//	Safety.GetDiagnostics(AddError:= AddError, a_ActiveEvents := a_ActiveEvents, w_index := w_errorindex);
//	Main_Fast.PowerMonitor.GetDiagnostics(AddError:= AddError, a_ActiveEvents := a_ActiveEvents, w_index := w_errorindex);
//	Main_Fast.InternalPowerSupply.GetDiagnostics(AddError:= AddError, a_ActiveEvents := a_ActiveEvents, w_index := w_errorindex);
//	Main_Fast.NeutralTransformer.GetDiagnostics(AddError:= AddError, a_ActiveEvents := a_ActiveEvents, w_index := w_errorindex);
//	Main_Fast.PowerStack.GetDiagnostics(AddError := AddError, a_ActiveEvents := a_ActiveEvents, w_index := w_errorindex);
//Main_Fast.Protectionsystems.GetDiagnostics(AddError := AddError, a_ActiveEvents := a_ActiveEvents, w_index := w_errorindex);
END_IF

//If larger than 0, error is existing
b_errorActive := GVL.b_NormalShutdownActive OR GVL.b_QuickshutdownActive OR GVL.b_EmergencyShutdownActive;

METHOD PUBLIC LimitTrigger
VAR_INPUT
	r_HighLimit				: REAL := 0;
	r_HighWarning			: REAL := 0;
	b_HighEnable			: BOOL := FALSE;
	r_LowLimit				: REAL := 0;
	r_LowWarning			: REAL := 0;
	b_LowEnable				: BOOL := FALSE;
	r_Hysteresis			: REAL := 0;
END_VAR

VAR_IN_OUT
	r_In					: REAL;
END_VAR

VAR_OUTPUT
	b_Warning				: BOOL;
	b_Fault					: BOOL;
END_VAR
IF b_HighEnable THEN
	IF r_IN >= r_HighLimit THEN
		b_Fault := TRUE;
	ELSIF r_IN < (r_HighLimit - r_Hysteresis) THEN
		b_fault := FALSE;
	END_IF
	IF r_IN >= r_HighWarning THEN
		b_warning := TRUE;
	ELSIF r_IN < (r_HighWarning - r_Hysteresis) THEN
		b_warning := FALSE;
	END_IF

END_IF

IF b_LowEnable THEN
	IF r_IN <= r_LowLimit THEN
		b_fault := TRUE;
	ELSIF r_IN > (r_LowLimit + r_Hysteresis) THEN
		b_fault := FALSE;
	END_IF
	IF r_IN <= r_LowWarning THEN
		b_warning := TRUE;
	ELSIF r_IN > (r_LowWarning + r_Hysteresis) THEN
		b_warning:= FALSE;
	END_IF
END_IF
END_METHOD

END_PROGRAM

// ---- POUs/ErrorHandling/FB_AddErrorST.TcPOU
FUNCTION_BLOCK FB_AddErrorST
VAR_INPUT
	in_b_ErrorTrig				: BOOL;
	in_t_TriggerTime			: TIME := T#0S;
	in_b_AutoClear				: BOOL := FALSE;
	in_e_ErrAckAccess			: eErrAckAccess := eErrAckAccess.VDL; //default full access required
	w_ID						: WORD;
	s_message					: STRING;
	e_sev						: eSeverity;
END_VAR
VAR_IN_OUT
	out_st_Error 				: ST_ErrorStruct;
END_VAR

VAR_OUTPUT
	b_out						: BOOL;
END_VAR

VAR
	sr_ErrorActive				: SR;
	bIsInitialized 				: BOOL := FALSE;	
	ton_FaultTriggerTime		: TON;
	rTRIG_Fault					: R_TRIG;
	fTRIG_Fault					: F_TRIG;
	rTRIG_Clear					: R_TRIG;
	
	
	i_Counter				: INT; 
END_VAR

IF NOT bIsInitialized THEN
    // The code that you want to be executed at the first cycle
		out_st_Error.s_ID		:= TO_STRING(w_ID);	
		out_st_Error.s_Message	:= TO_STRING(s_Message);
		out_st_Error.s_Severity	:= TO_STRING(e_Sev);
END_IF

ton_FaultTriggerTime(IN:= in_b_ErrorTrig, PT:= in_t_TriggerTime);
sr_ErrorActive(SET1:= ton_FaultTriggerTime.Q, Q1=>out_st_error.b_ErrorActive);
b_out := sr_ErrorActive.Q1;

sr_ErrorActive.RESET := SEL( errorhandling.e_access>=in_e_ErrAckAccess,0,Errorhandling.b_ResetError);

CASE e_sev OF
		eSeverity.Warning 			: GVL.b_WarningActive := b_out;
		eSeverity.Normalshutdown 	: GVL.b_NormalshutdownActive := b_out;
		eSeverity.Quickshutdown 	: GVL.b_QuickShutdownActive := b_out;
		eSeverity.EmergencyShutdown	: GVL.b_EmergencyShutdownActive := b_out;
END_CASE


//CLEARING EVENTS
rTRIG_Fault(CLK:= b_out);
fTRIG_Fault(CLK:= b_out);
rTRIG_Clear(CLK:= ErrorHandling.b_ClearEvents OR SEL(in_b_autoClear,FALSE, errorhandling.ton_AutoResetClear.Q) );

IF rTRIG_Clear.Q AND NOT b_out THEN
	out_st_Error.s_DateError 	:= '';
	out_st_Error.s_TimeError 	:= '';
	out_st_Error.s_TimeCleared	:= '';
END_IF

IF rTRIG_Fault.Q THEN
	out_st_Error.s_DateError := GVL.s_SystemDate;
	out_st_Error.s_TimeError := GVL.s_SystemTime;
	out_st_Error.s_TimeCleared	:= '';
	
ELSIF fTrig_Fault.Q THEN
	out_st_Error.s_TimeCleared	:= GVL.s_SystemTime;
END_IF

bIsInitialized := TRUE;

END_FUNCTION_BLOCK

// ---- POUs/FunctionBlocks/fbDwordToReal.TcPOU
FUNCTION_BLOCK fbDwordToReal
VAR_INPUT
	in_B0					: BYTE ;
	in_B1					: BYTE ;
	in_B2					: BYTE ;
	in_B3					: BYTE ;
	in_r_Res				: REAL ;
	in_i_Offset				: INT ;
END_VAR
VAR_OUTPUT
	out_r_Value				: REAL ;
END_VAR
VAR
	di_AddedValue			: DINT;
	r_Signed				: REAL;
	r_ResolutionResolved	: REAL;
END_VAR

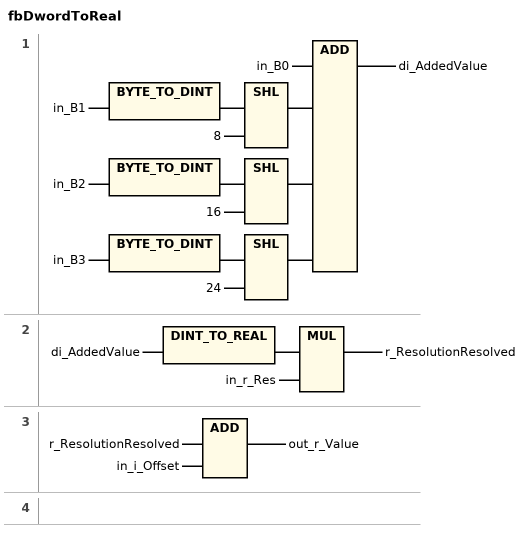
// NETWORK 1
di_AddedValue := in_B0 + SHL(BYTE_TO_DINT(in_B1), 8) + SHL(BYTE_TO_DINT(in_B2), 16) + SHL(BYTE_TO_DINT(in_B3), 24);

// NETWORK 2
r_ResolutionResolved := DINT_TO_REAL(di_AddedValue) * in_r_Res;

// NETWORK 3
out_r_Value := r_ResolutionResolved + in_i_Offset;

// NETWORK 4

END_FUNCTION_BLOCK

// ---- POUs/FunctionBlocks/fbRealToDWord.TcPOU
FUNCTION_BLOCK fbRealToDWord
VAR_INPUT
	in_r_Value				: REAL ;
	in_r_Res				: REAL ;
	in_i_Offset				: INT ;
END_VAR
VAR_OUTPUT
	out_B0					: BYTE ;
	out_B1					: BYTE ;
	out_B2					: BYTE ;
	out_B3					: BYTE ;
END_VAR
VAR
	dw_AddedValue			: DWORD;
	r_ResolutionResolved	: REAL;
	r_OffsetSolved			: REAL;
END_VAR

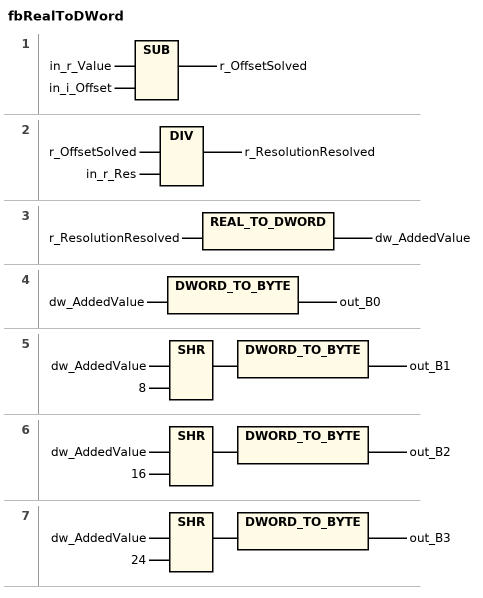
// NETWORK 1
r_OffsetSolved := in_r_Value - in_i_Offset;

// NETWORK 2
r_ResolutionResolved := r_OffsetSolved / in_r_Res;

// NETWORK 3
dw_AddedValue := REAL_TO_DWORD(r_ResolutionResolved);

// NETWORK 4
out_B0 := DWORD_TO_BYTE(dw_AddedValue);

// NETWORK 5
out_B1 := DWORD_TO_BYTE(SHR(dw_AddedValue, 8));

// NETWORK 6
out_B2 := DWORD_TO_BYTE(SHR(dw_AddedValue, 16));

// NETWORK 7
out_B3 := DWORD_TO_BYTE(SHR(dw_AddedValue, 24));

END_FUNCTION_BLOCK

// ---- POUs/FunctionBlocks/fbRealToWord.TcPOU
FUNCTION_BLOCK fbRealToWord
VAR_INPUT
	in_r_Value				: REAL ;
	in_r_Res				: REAL ;
	in_i_Offset				: INT ;
END_VAR
VAR_OUTPUT
	out_B0					: BYTE ;
	out_B1					: BYTE ;
END_VAR
VAR
	w_AddedValue			: WORD;
	r_ResolutionResolved	: REAL;
	r_OffsetSolved			: REAL;
END_VAR

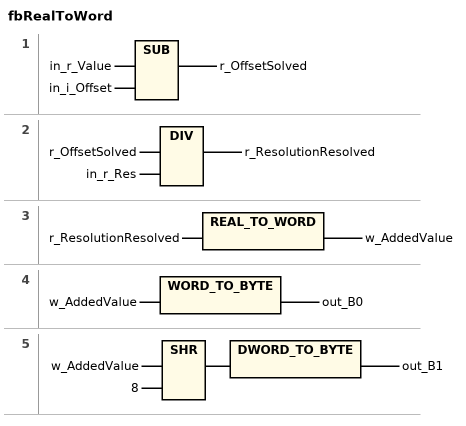
// NETWORK 1
r_OffsetSolved := in_r_Value - in_i_Offset;

// NETWORK 2
r_ResolutionResolved := r_OffsetSolved / in_r_Res;

// NETWORK 3
w_AddedValue := REAL_TO_WORD(r_ResolutionResolved);

// NETWORK 4
out_B0 := WORD_TO_BYTE(w_AddedValue);

// NETWORK 5
out_B1 := DWORD_TO_BYTE(SHR(w_AddedValue, 8));

END_FUNCTION_BLOCK

// ---- POUs/FunctionBlocks/fbWordToReal.TcPOU
FUNCTION_BLOCK fbWordToReal
VAR_INPUT
	in_B0					: BYTE ;
	in_B1					: BYTE ;
	in_r_Res				: REAL ;
	in_i_Offset				: INT ;
END_VAR
VAR_OUTPUT
	out_r_Value				: REAL ;
END_VAR
VAR
	dw_AddedValue			: DWORD;
	r_ResolutionResolved	: REAL;
END_VAR

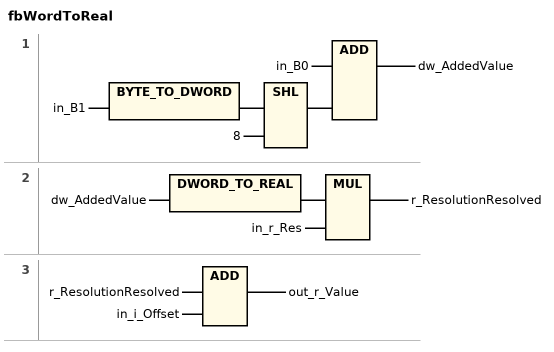
// NETWORK 1
dw_AddedValue := in_B0 + SHL(BYTE_TO_DWORD(in_B1), 8);

// NETWORK 2
r_ResolutionResolved := DWORD_TO_REAL(dw_AddedValue) * in_r_Res;

// NETWORK 3
out_r_Value := r_ResolutionResolved + in_i_Offset;

END_FUNCTION_BLOCK

// ---- POUs/MonitoringControl/FB_ControlManager.TcPOU
FUNCTION_BLOCK FB_ControlManager

VAR_OUTPUT PERSISTENT
	Hardsettings_persistent					: ST_HardSettings; 
	Softsettings_persistent					: ST_Softsettings;
END_VAR

VAR_OUTPUT
	control									: ST_ControlVars;
	Operation								: ST_OperationVars;
END_VAR

VAR
	IoT							: FB_ControlSource_IoT;	
	PNController				: FB_PNController;
	{ attribute 'TcHmiSymbol.Show' }
	b_SettingsChanged			: BOOL;				
END_VAR

VAR_IN_OUT CONSTANT
	{ attribute 'TcHmiSymbol.Hide' }
	monitor						: ST_SystemControl_FromSystem;
END_VAR

//instantiate fbs 
hmi(monitor:=monitor, PLCsettingsHard:= Hardsettings_persistent, PLCsettingsSoft :=SoftSettings_persistent);
PNController(monitor := monitor);
Iot(monitor:=monitor);

ControlSourceSelector();



//refresh HMI data --> future work make on change and asynchronous java in hmi

METHOD PROTECTED ControlSourceSelector

VAR_OUTPUT
	b_Busy					: BOOL;
	b_Error					: BOOL;
END_VAR

VAR
	
	softsettingsTemp				: ST_SoftSettings;
	controlTemp						: ST_ControlVars;
	
	rtrig_WritePersistent		: R_TRIG;
	fb_WritePersistentData		: WritePersistentData;
END_VAR
//Choosing the control source always requires the HMI
IF HMI.controlvars.control.b_ActivateSettings THEN
	Hardsettings_persistent.setup.e_ControlSource := HMI.Controlvars.hardSettings.setup.e_ControlSource;
END_IF


CASE Hardsettings_persistent.setup.e_ControlSource OF
	eControlSources.Local: // HMI
		softsettingsTemp 	:= HMI.controlvars.SoftSettings;
		Operation			:= HMI.controlvars.Operation;
	eControlSources.ExternalController: // HMI
		softsettingsTemp 	:= PnController.SoftSettings;
		Operation			:= PNController.Operation;	
		controlTemp			:= PNController.control;
	eControlSources.IoT:	//IOT
		softsettingsTemp 	:= IoT.SoftSettings; // Only local HMI can adjust recipe and thus persistent values.
		Operation			:= IoT.operation;
		controlTemp			:= IoT.control;
END_CASE

// WRITE PRIORITY DATA
control.b_start := HMI.controlvars.control.b_start OR controltemp.b_start;
control.b_Shutdown := HMI.controlvars.control.b_Shutdown OR controltemp.b_Shutdown;
control.b_ClearHistory := HMI.controlvars.control.b_ClearHistory OR controltemp.b_ClearHistory;
control.b_Reset := HMI.controlvars.control.b_Reset OR controltemp.b_Reset;
control.b_ActivateSettings := HMI.controlvars.control.b_ActivateSettings OR controltemp.b_ActivateSettings;
control.b_Reboot:= HMI.controlvars.control.b_Reboot OR controltemp.b_Reboot;
control.b_EMstop:= HMI.controlvars.control.b_EMstop OR controltemp.b_EMstop;
control.b_ResetVDL := HMI.controlvars.control.b_ResetVDL OR Iot.control.b_ResetVDL;


//WRITE PERSISTENT DATA
rtrig_WritePersistent(CLK:=HMI.controlvars.control.b_ActivateSettings);
IF rtrig_WritePersistent.Q THEN
	Hardsettings_persistent := HMI.controlvars.HardSettings;
	Softsettings_persistent	:= softsettingsTemp;
	fb_WritePersistentData(NETID := '', PORT:= 851, START:=TRUE, TMOUT := T#1S);
ELSE
	fb_WritePersistentData(START := FALSE);
END_IF

b_Busy := fb_WritePersistentData.BUSY;
b_Error := fb_WritePersistentData.ERR;
END_METHOD

END_FUNCTION_BLOCK

// ---- POUs/MonitoringControl/ProfinetController/FB_PNController.TcPOU
FUNCTION_BLOCK FB_PNController
VAR_OUTPUT
	{ attribute 'TcHmiSymbol.ShowRecursively' }
	control							: ST_ControlVars;	//1 module
	Operation						: ST_OperationVars;	//4 modules
	SoftSettings					: ST_SoftSettings;	//4 modules
	get								: ST_PNController_get;
END_VAR

VAR_IN_OUT CONSTANT
	{ attribute 'TcHmiSymbol.Hide' }
	monitor								: ST_SystemControl_FromSystem;
END_VAR

VAR
	CouplerState	AT %I*		:	WORD;	
	CouplerDiag		AT %I*		:	WORD;	

	GeneralInputs 	AT %I*		:	ST_PNInput_General;
	GeneralOutputs	AT %Q*		:	ST_PNOutput_General;
	
	BatteryInputs 	AT %I*		:	ST_PNInput_Battery;
	BatteryOutputs 	AT %Q*		:	ST_PNOutput_Battery;
	
	OutputFieldOutputs AT %Q*	:	ST_PNOutput_OutputField;
	
	InputFieldInputs	AT %I* 	:	ST_PNInput_InputField;
	InputFieldOutputs	AT %Q* 	:	ST_PNOutput_InputField;
	
	PowerStackInputs	AT %I* 	:	ST_PNInput_PowerStack;
	PowerStackOutputs	AT %Q* 	:	ST_PNOutput_PowerStack;	
	
	PeakShaveBoxInputs	AT %I* 	:	ST_PNInput_PeakShaveBox;
	PeakShaveBoxOutputs	AT %Q* 	:	ST_PNOutput_PeakShaveBox;
	
	ZPTOutputs			AT %Q* 	:	ST_PNOutput_ZPT;
	
END_VAR

VAR_INPUT
	b_enableControl	:	BOOL;
	b_enableMonitor	:	BOOL;
END_VAR


MapGeneralData	(Input := GeneralInputs, 		Output => Generaloutputs		);
MapBatteryData	(Input := BatteryInputs,		Output => BatteryOutputs		);
MapOutputField	(								Output => OutputFieldOutputs	);
MapInputField	(Input := InputFieldInputs, 	Output => InputFieldOutputs		);
MapPowerStack	(Input := PowerSTackInputs, 	Output => PowerStackOutputs		);
MapPeakShaveBox	(Input := PeakShaveBoxInputs, 	Output => PeakShaveBoxOutputs	);
MapZPT			(								Output => ZPTOutputs			);

PNCouplerDiagnostics (DevState:=CouplerState, DevDiag := CouplerDiag);

METHOD DwordToReal : REAL
VAR_INPUT
	InputVar			:	DWORD;
	b_InputSigned		:	BOOL;
	Stepsize			:	WORD;
end_var
DwordToReal := 1;

IF b_inputSigned AND InputVar.31 THEN
	DwordToReal := -1;
	InputVar.31 := FALSE;
END_IF

DwordToReal := DwordToReal * DWORD_TO_REAL(InputVar)/Stepsize;
END_METHOD

METHOD EMStop : BOOL
VAR_INPUT
END_VAR

//?

EMStop := true;
END_METHOD

METHOD GetDiagnostics 
VAR_IN_OUT
	AddError		: ARRAY [*] OF FB_AddErrorST;
	a_ActiveEvents	: ARRAY [*] OF ST_ErrorStruct;
	w_Index			: WORD;
END_VAR

VAR_OUTPUT
	b_errorActive	: BOOL;
	b_warningActive	: BOOL;
END_VAR

VAR
	by_errCt	: BYTE;
	by_warnCt	: BYTE;
	w_ID		: WORD;
END_VAR
	(*PN coupler data configuration fault*)	AddError[w_Index](
			in_b_ErrorTrig			:= Get.Events.b_DataConfigurationFault
			out_ST_Error			:= a_ActiveEvents[w_Index],
			w_ID					:= 1 + w_ID,
			s_Message				:= 'Profinet Data configuration fault',
			e_sev					:= eSeverity.Warning,	
			in_b_AutoClear			:= FALSE,
			//in_e_ErrAckAccess		:= TRUE,
			);
		IF AddError[w_Index].b_out THEN by_warnCt := by_warnCt + 1; END_IF;
		w_Index := w_Index +1;
		
	(*Profinet coupler device fault*)	AddError[w_Index](
			in_b_ErrorTrig			:= Get.Events.b_DeviceFault,
			out_ST_Error			:= a_ActiveEvents[w_Index],
			w_ID					:= 2 + w_ID,
			s_Message				:= 'Profinet control device fault',
			e_sev					:= eSeverity.Warning,	
			in_b_AutoClear			:= FALSE,
			//in_e_ErrAckAccess		:= TRUE,
			);
		IF AddError[w_Index].b_out THEN by_warnCt := by_warnCt + 1; END_IF;
		w_Index := w_Index +1;
	
	(*Profinet heartbeat lost*)	AddError[w_Index](
			in_b_ErrorTrig			:= Get.Events.b_HeartBeatLost,
			out_ST_Error			:= a_ActiveEvents[w_Index],
			w_ID					:= 3 + w_ID,
			s_Message				:= 'Profinet control watchdog fault',
			e_sev					:= eSeverity.QuickShutdown,	
			in_b_AutoClear			:= FALSE,
			//in_e_ErrAckAccess		:= TRUE,
			);
		IF AddError[w_Index].b_out THEN by_warnCt := by_warnCt + 1; END_IF;
		w_Index := w_Index +1;
		
	(*Profinet control network config fault*)	AddError[w_Index](
			in_b_ErrorTrig			:= Get.Events.b_NetworkConfigurationFault,
			out_ST_Error			:= a_ActiveEvents[w_Index],
			w_ID					:= 4 + w_ID,
			s_Message				:= 'Profinet control network config fault',
			e_sev					:= eSeverity.Warning,	
			in_b_AutoClear			:= FALSE,
			//in_e_ErrAckAccess		:= TRUE,
			);
		IF AddError[w_Index].b_out THEN by_warnCt := by_warnCt + 1; END_IF;
		w_Index := w_Index +1;
END_METHOD

METHOD HeartBeat : BOOL
VAR_INPUT
	ui_HeartBeatInput		:	UINT	:=	0;
END_VAR

VAR_OUTPUT
	ui_HeartBeatOutput		:	UINT	:=	0;
END_VAR

VAR_INST
	HeartBeatOutputIncTimer		:	TON		:=	(PT := T#500MS);
	HeartBeatInputCheckTimer	:	TON		:=	(PT := T#1S);
	ui_StoredInputValue			:	UINT	:= 	0;
END_VAR

//output value increments every second. Remote party should check if this happens
HeartBeatOutputIncTimer ( in := NOT HeartBeatOutputIncTimer.Q);
IF HeartBeatOutputIncTimer.Q THEN
	ui_HeartBeatOutput := ui_HeartBeatOutput +1;
END_IF

//Input value has to change every second as well.
//if stored and Current values are equal, start counting.
HeartBeatInputCheckTimer(in:= (ui_StoredInputValue = ui_HeartBeatInput));
ui_StoredInputValue := ui_HeartBeatInput;
get.events.b_HeartBeatLost := HeartBeatInputCheckTimer.Q;
END_METHOD

METHOD IntToReal : Real
VAR_INPUT
	in		:	INT;
	Scale	:	UINT := 10;
END_VAR
intToReal := INT_TO_REAL(in)/Scale;
END_METHOD

METHOD MapBatteryData : BOOL
VAR_INPUT
	Input	:	ST_PNInput_Battery;
END_VAR

VAR_OUTPUT
	Output	:	ST_PNOutput_Battery;
END_VAR


VAR

END_VAR
//Fill output data
IF b_enableMonitor THEN
	Output.w_Status.0	:=	Monitor.battery.BattInfo.ui_BMS_PowerOnStatus = ePowerOnStatus.On;	
	Output.w_Status.1	:=	Monitor.battery.BattInfo.ui_BMS_Status = eBMS_Status.Init;
	Output.w_Status.2	:=	Monitor.battery.BattInfo.ui_BMS_Status = eBMS_Status.Normal;
	Output.w_Status.3	:=	Monitor.battery.BattInfo.ui_BMS_Status = eBMS_Status.FullCharge;
	Output.w_Status.4	:=	Monitor.battery.BattInfo.ui_BMS_Status = eBMS_Status.FullDischarge;
	Output.w_Status.5	:=	Monitor.battery.BattInfo.ui_BMS_Status = eBMS_Status.Warning;
	Output.w_Status.6	:=	Monitor.battery.BattInfo.ui_BMS_Status = eBMS_Status.Fault;
	
	Output.w_Warnings.0 := Monitor.battery.events.b_OVER_TEMP_WARNING;	
	Output.w_Warnings.1 := Monitor.battery.events.b_UNDER_TEMP_WARNING;			
	Output.w_Warnings.2 := Monitor.battery.events.b_OVER_CHARGE_CURRENT_WARNING;	
	Output.w_Warnings.3 := Monitor.battery.events.b_OVER_DISCHARGE_CURRENT_WARNING;
	Output.w_Warnings.4 := Monitor.battery.events.b_OVER_VOLT_WARNING;		
	Output.w_Warnings.5 := Monitor.battery.events.b_UNDER_VOLT_WARNING;		
	Output.w_Warnings.6 := Monitor.battery.events.b_UNDER_SOC_MIN_WARNING;		
	Output.w_Warnings.7 := Monitor.battery.events.b_OVER_SOC_MAX_WARNING;			
	Output.w_Warnings.8 := Monitor.battery.events.b_VOLTAGE_IMBALANCE_WARNING;
	Output.w_Warnings.9 := Monitor.battery.events.b_TEMPERATURE_IMBALANCE_WARNING;
	Output.w_Warnings.10 := Monitor.battery.events.b_CURRENT_IMBALANCE_WARNING;
	Output.w_Warnings.11 := Monitor.battery.events.b_OTHER_WARNING;	
	Output.w_Warnings.12 := Monitor.battery.events.b_CONFIGURATION_WARNING;
	
	Output.w_Faults.0 := Monitor.battery.Events.b_COMMUNICATION_ERROR;			
	Output.w_Faults.1 := Monitor.battery.events.b_OVER_TEMP_ALARM;					
	Output.w_Faults.2 := Monitor.battery.events.b_UNDER_TEMP_ALARM;			
	Output.w_Faults.3 := Monitor.battery.events.b_OVER_CHARGE_CURRENT_ALARM;		
	Output.w_Faults.4 := Monitor.battery.events.b_OVER_DISCHARGE_CURRENT_ALARM;	
	Output.w_Faults.5 := Monitor.battery.events.b_OVER_VOLT_ALARM;						
	Output.w_Faults.6 := Monitor.battery.events.b_UNDER_VOLT_ALARM;					
	Output.w_Faults.7 := Monitor.battery.events.b_UNDER_SOC_MIN_ALARM;				
	Output.w_Faults.8 := Monitor.battery.events.b_OVER_SOC_MAX_ALARM;				
	Output.w_Faults.9 := Monitor.battery.events.b_TEMPERATURE_IMBALANCE_ALARM;	
	Output.w_Faults.10 := Monitor.battery.events.b_CONTACTOR_ERROR;				
	Output.w_Faults.11 := Monitor.battery.events.b_FAN_ERROR;						
	Output.w_Faults.12 := Monitor.battery.events.b_GROUND_FAULT;					
	Output.w_Faults.13 := Monitor.battery.events.b_OPEN_DOOR_ERROR;					
	Output.w_Faults.14 := Monitor.battery.events.b_OTHER_ALARM;								
	Output.w_Faults.15 := Monitor.battery.events.b_CONFIGURATION_ALARM;			
				
	Output.ui_SOC 							:= RealToUint(	In	:=	monitor.battery.Battinfo.r_SOC, 	Scale	:=	10);
	Output.ui_SOH 							:= RealToUint(	In	:=	monitor.battery.Battinfo.r_SOH, 	Scale	:=	10);
	Output.ui_DClinkVoltage 				:= RealToUint(	In	:=	monitor.battery.Battinfo.r_SystemVoltage, Scale	:=	10);				
	Output.i_DClinkCurrent 					:= RealToint (	In	:=	monitor.battery.Battinfo.r_SystemCurrent, Scale	:=	10);
	Output.ui_MaxAllowedDischargeCurrent 	:= RealToUint (	In	:=	monitor.battery.Battinfo.r_MaxDischargeCurrentAllowed, Scale	:=	10); 	
	Output.ui_MaxAllowedChargeCurrent 		:= RealToUint (	In	:=	monitor.battery.Battinfo.r_MaxchargeCurrentAllowed,	Scale	:=	10); 		
	Output.i_MinCellTemperature 			:= RealToint (	In	:=	monitor.battery.Battinfo.ar_CellTemperature[0] , Scale	:=	10); 	
	Output.i_MaxCellTemperature				:= RealToint (	In	:=	monitor.battery.Battinfo.ar_CellTemperature[2], Scale	:=	10); 										                                               
	Output.ui_RemainingChargeEnergy 		:= RealToUint(	In	:=	monitor.battery.Battinfo.r_RemainingChargeEnergy, Scale	:=	10);
	Output.ui_RemainingDischargeEnergy 		:= RealToUint(	In	:=	monitor.battery.Battinfo.r_RemainingDischargeEnergy, Scale	:=	10);
	Output.ui_HistAccChargeEnergy_high		:= UDINT_TO_UINT(SHR(RealToUdint(	In	:=	monitor.battery.Battinfo.r_HistAccChargeEnergy, Scale	:=	10), 16));
	Output.ui_HistAccChargeEnergy_low		:= UDINT_TO_UINT(RealToUdint(	In	:=	monitor.battery.Battinfo.r_HistAccChargeEnergy, Scale	:=	10));
	Output.ui_HistAccDischargeEnergy_high 	:= UDINT_TO_UINT(SHR(RealToUDint(	In	:=	monitor.battery.Battinfo.r_HistAccDischargeEnergy, Scale	:=	10), 16));
	Output.ui_HistAccDischargeEnergy_low 	:= UDINT_TO_UINT(RealToUDint(	In	:=	monitor.battery.Battinfo.r_HistAccDischargeEnergy, Scale	:=	10));
END_IF


//process input data
IF NOT get.events.b_HeartBeatLost AND b_enableControl THEN
	SoftSettings.system.r_SocMin	:=	LIMIT(0, UINT_TO_REAL(Input.ui_SocMinLimit)/10, 100);
	SoftSettings.system.r_SocMax	:=	LIMIT(0, UINT_TO_REAL(Input.ui_SocMinLimit)/10, 100);
END_IF
END_METHOD

METHOD MapGeneralData : BOOL
VAR_INPUT
	Input	:	ST_PNInput_General;
END_VAR

VAR_OUTPUT
	Output	:	ST_PNOutput_General;
END_VAR

VAR


END_VAR
//First check heartbeat status
HeartBeat(ui_HeartBeatInput := input.ui_HeartBeat, ui_HeartBeatOutput => output.ui_HeartBeatOut);


IF b_enableMonitor THEN
	Output.w_SystemState		:=	Monitor.system.e_State;
	Output.w_SystemStatus.0		:= 	Monitor.protections.Insulation.b_Enabled;
	Output.w_SystemStatus.1		:=	b_enableControl;	
	Output.w_SystemStatus.8		:=	Monitor.system.e_EarthingSystem = eEarthingSystems.TNS;
	Output.w_SystemStatus.9		:=	Monitor.system.e_EarthingSystem = eEarthingSystems.TNC;
	Output.w_SystemStatus.10	:=	Monitor.system.e_EarthingSystem = eEarthingSystems.IT;
	
	Output.w_SystemWarnings.0	:=	Monitor.protections.FireDetection.CODetectors.State = eCOAlarmStatus.WarningLevel1;
	Output.w_SystemWarnings.1	:=	Monitor.protections.FireDetection.CODetectors.State = eCOAlarmStatus.WarningLevel2;
	Output.w_SystemWarnings.2	:=	Monitor.protections.Insulation.b_Warning;
	Output.w_SystemWarnings.3	:=	Monitor.protections.MRCDB.b_prewarning;
	Output.w_SystemWarnings.8	:=	Monitor.protections.FireDetection.Events.SmokeDetFault;
	Output.w_SystemWarnings.9	:=	Monitor.protections.FireDetection.Events.CODetFault;
	Output.w_SystemWarnings.10	:=	NOT Monitor.protections.Surge.b_Type12_OK;
	Output.w_SystemWarnings.11	:=	NOT Monitor.protections.Surge.b_Type3_OK;
	Output.w_SystemWarnings.12	:=	NOT Monitor.enclosure.doors.b_ControlPanelDoorClosed;
	Output.w_SystemWarnings.13	:=	NOT Monitor.enclosure.doors.b_ClientpanelDoorClosed;
	
	Output.w_SystemFaults.0		:=	Monitor.protections.FireDetection.Events.SmokeDetAlarm;
	Output.w_SystemFaults.1		:=	Monitor.protections.FireDetection.Events.CODetAlarm;
	Output.w_SystemFaults.2		:=	NOT Monitor.safety.b_InsulationMonitorOK;
	Output.w_SystemFaults.3		:=	NOT Monitor.safety.b_MRCDBOK;
	Output.w_SystemFaults.8		:=	NOT Monitor.safety.b_InverterDoorOK;
	
	Output.w_CoolingSystemStatus.0	:=	Monitor.Cooling.CoolingSystemMode = eConditioningStates.OFF;
	Output.w_CoolingSystemStatus.1	:=	Monitor.Cooling.CoolingSystemMode = eConditioningStates.EnclosureConditioning;
	Output.w_CoolingSystemStatus.2	:=	Monitor.Cooling.CoolingSystemMode = eConditioningStates.BatteryConditioning;
	Output.w_CoolingSystemStatus.3	:=	Monitor.Cooling.CoolingSystemMode = eConditioningStates.DeHum;
	Output.w_CoolingSystemStatus.4	:=	(Monitor.Cooling.CoolingSystemMode = eConditioningStates.InverterPowerMode) OR
										(Monitor.Cooling.CoolingSystemMode = eConditioningStates.InverterZPTStartup) ;
	Output.w_CoolingSystemStatus.8	:=	Monitor.Cooling.HeatPumpStatus = eHeatPumpState.Active_Cooling;
	Output.w_CoolingSystemStatus.9	:=	Monitor.Cooling.HeatPumpStatus = eHeatPumpState.Active_Heating;
	
	Output.w_CoolingSystemWarnings.0	:=	Monitor.Cooling.Events.b_SystemOvertemperatureWarning;
	Output.w_CoolingSystemWarnings.1	:=	Monitor.Cooling.Events.b_SystemUndertemperatureWarning;
	Output.w_CoolingSystemWarnings.2	:=	Monitor.Cooling.Events.b_CoolingLoopIdlePressureWarning;
	Output.w_CoolingSystemWarnings.3	:=	Monitor.Cooling.Events.b_HeatpumpWarning;
	
	Output.w_CoolingSystemFaults.0	:=	Monitor.Cooling.Events.b_CoolingSystemFuseFailure;
	Output.w_CoolingSystemFaults.1	:=	Monitor.Cooling.Events.b_BattLoopValveStuck OR 
										Monitor.Cooling.Events.b_FancoilLoopValveStuck OR 
										Monitor.Cooling.Events.b_InverterLoopValveStuck;
	Output.w_CoolingSystemFaults.2	:=	Monitor.Cooling.Events.b_CoolingLoopIdlePressureError;									
	Output.w_CoolingSystemFaults.3	:=	Monitor.Cooling.Events.b_HeatpumpError;
		
	Output.w_InternalSupplyStatus.0	:=	Monitor.internalpsu.b_24VdcAvailable;
	Output.w_InternalSupplyStatus.1	:=	Monitor.internalpsu.b_400VACAvailable;
	Output.w_InternalSupplyStatus.2	:=	Monitor.internalpsu.b_HVDCAvailable;
	Output.w_InternalSupplyStatus.3	:=	Monitor.internalpsu.UPS.b_SystemOnBattery;
	
	Output.w_InternalSupplyWarnings.0 :=	Monitor.internalpsu.UPS.Events.b_BatteryLowWarning;
	
	Output.w_InternalSupplyFaults.0 :=	Monitor.internalpsu.UPS.Events.b_BatteryLowError;
	Output.w_InternalSupplyFaults.1 :=	Monitor.internalpsu.Events.b_ACPSUFault;
	Output.w_InternalSupplyFaults.2 :=	Monitor.internalpsu.Events.b_CEEInputFuseTripped;
	Output.w_InternalSupplyFaults.3 :=	Monitor.internalpsu.Events.b_DCPSUFault;
	Output.w_InternalSupplyFaults.4 :=	Monitor.internalpsu.Events.b_GridInputFuseTripped;
END_IF

IF NOT get.events.b_HeartBeatLost AND b_enableControl THEN
	Control.b_start 								:= Input.W_Control.0;
	Control.b_stop									:= Input.W_Control.1;
	Control.b_shutdown 								:= Input.W_Control.2;
	Control.b_Reset 								:= Input.W_Control.3;
	Control.b_EMstop 								:= Input.W_Control.4;
	Control.b_ActivateSettings						:= Input.W_Control.5;
	Softsettings.system.b_AutomaticSwitching		:= Input.W_Control.6;
	Softsettings.system.b_EnableConditioningMode	:= Input.W_Control.7;
	Softsettings.system.b_StartDehumidifyingCycle	:= Input.W_Control.8;
END_IF
END_METHOD

METHOD MapInputField : BOOL
VAR_INPUT
	Input	:	ST_PNInput_InputField;
END_VAR

VAR_OUTPUT
	Output	:	ST_PNOutput_InputField;
END_VAR

//Fill output data
IF b_enableMonitor THEN
	Output.w_Status.0	:=	Monitor.ACswitchgear.b_InputContactorfb;
	Output.w_Status.1	:=	Monitor.ACswitchgear.b_InputMCCBfb;
	Output.w_Status.2	:=	Monitor.ACswitchgear.b_InputSynchronizerfb;
	
	Output.w_Warnings.0	:=	Monitor.ACswitchgear.b_InputMCCBShuntOK;
	Output.w_Warnings.1	:=	Monitor.powermonitor.events.b_MBCommWarning OR 
							Monitor.powermonitor.events.b_MBTimeoutWarning OR 
							Monitor.powermonitor.events.b_EL3443Warning;
	Output.w_Warnings.3	:=	Monitor.protections.OvercurrentProtection.b_InputWarning;
	
	Output.w_Faults.0	:=	Monitor.protections.OvercurrentProtection.b_InputAlarm;
	Output.w_Faults.1	:=	Monitor.powermonitor.events.b_MBCommError OR Monitor.powermonitor.events.b_EL3443Error;

	Output.i_ActivePower 			:=	RealToint (	In	:= Monitor.powermonitor.OutputField.r_ActivePower, 	Scale	:=	10);
	Output.i_ReactivePower 			:=	RealToint (	In	:= Monitor.powermonitor.OutputField.r_ReactivePower, Scale	:=	10);
	Output.ui_frequency				:=	RealToUint(	In	:= Monitor.powermonitor.OutputField.r_Frequency, 	Scale	:=	10);
	Output.ui_VoltageL1N			:=	RealToUint(	In	:= Monitor.powermonitor.OutputField.r_PhaseVoltage[1], Scale	:=	10);
	Output.ui_VoltageL2N			:=	RealToUint(	In	:= Monitor.powermonitor.OutputField.r_PhaseVoltage[2], Scale	:=	10);
	Output.ui_VoltageL3N			:=	RealToUint(	In	:= Monitor.powermonitor.OutputField.r_PhaseVoltage[3], Scale	:=	10);
	Output.ui_VoltageL1L2			:=	RealToUint(	In	:= Monitor.powermonitor.OutputField.r_LineVoltage[1], Scale	:=	10);
	Output.ui_VoltageL2L3			:=	RealToUint(	In	:= Monitor.powermonitor.OutputField.r_LineVoltage[2], Scale	:=	10);
	Output.ui_VoltageL3L1			:=	RealToUint(	In	:= Monitor.powermonitor.OutputField.r_LineVoltage[3], Scale	:=	10);
	Output.i_CurrentL1				:=	RealToint (	In	:= Monitor.powermonitor.OutputField.r_Current[1], 	Scale	:=	10);
	Output.i_CurrentL2				:=	RealToint (	In	:= Monitor.powermonitor.OutputField.r_Current[2], 	Scale	:=	10);
	Output.i_CurrentL3				:=	RealToint (	In	:= Monitor.powermonitor.OutputField.r_Current[3], 	Scale	:=	10);
	Output.i_CurrentN				:=	RealToint (	In	:= Monitor.powermonitor.OutputField.r_Current[4], 	Scale	:=	10);
	Output.ui_TotalEnergyConsumed_high	:= UDINT_TO_UINT(SHR(RealToUdint(	In	:=	monitor.powermonitor.InputField.r_EnergyConsumed, Scale	:=	10), 16));
	Output.ui_TotalEnergyConsumed_low	:= UDINT_TO_UINT(RealToUdint(	In	:=	monitor.powermonitor.InputField.r_EnergyConsumed, Scale	:=	10));
	Output.ui_TotalEnergySupplied_high 	:= UDINT_TO_UINT(SHR(RealToUdint(	In	:=	monitor.powermonitor.InputField.r_EnergySupplied, Scale	:=	10), 16));
	Output.ui_TotalEnergySupplied_low 	:= UDINT_TO_UINT(RealToUdint(	In	:=	monitor.powermonitor.InputField.r_EnergySupplied, Scale	:=	10));
	
END_IF

IF NOT get.events.b_HeartBeatLost AND b_enableControl THEN
	Operation.inputgenset.b_ManualStart 					:= Input.w_Control.0;
	Operation.inputgrid.b_ForceClose						:= Input.w_Control.1;	//Maybe unneccessary to write both?
	Operation.InputGenset.b_ForceClose						:= Input.w_Control.1;
	Operation.inputgrid.b_SyncClose							:= Input.w_Control.2;	//Maybe unneccessary to write both?
	Operation.InputGenset.b_SyncClose						:= Input.w_Control.2;
	SoftSettings.inputgrid.b_AutomaticMainsFailureRestart	:= Input.w_Control.3;
	
	SoftSettings.inputgrid.setpointTimeslot1.r_FeedInCurrentLimitSoft 	:= UintToReal(in:=Input.ui_FeedInCurrentLimit, Scale := 10);
	SoftSettings.inputgrid.setpointTimeslot1.r_SupplyCurrentLimitSoft 	:= UintToReal(in:=Input.ui_FeedOutCurrentLimit, Scale := 10);
	SoftSettings.inputgrid.setpointTimeslot1.r_IdleChargePower			:= UintToReal(in:=Input.ui_IdleChargePower, Scale := 10);
	SoftSettings.inputgrid.setpointTimeslot1.r_SocTarget				:= UINT_TO_REAL(Input.ui_SocTarget);
	SoftSettings.inputgenset.Conditions.by_SoCStart						:= UINT_TO_BYTE(Input.ui_SOCStart);	
	SoftSettings.inputgenset.Conditions.by_SoCStop						:= UINT_TO_BYTE(Input.ui_SOCStop);
	SoftSettings.inputgenset.Conditions.r_BatteryOverloadStart			:= UintToReal(In := Input.ui_BatterOverloadStart, Scale := 10);
	SoftSettings.inputgenset.Conditions.r_BatteryOverloadStop			:= UintToReal(In := Input.ui_BatteryOverloadStop, Scale := 10);
END_IF
END_METHOD

METHOD MapOutputField : BOOL
VAR_INPUT
	//Input	:	ST_PNInput_OutputField;
END_VAR

VAR_OUTPUT
	Output	:	ST_PNOutput_OutputField;
END_VAR

VAR

END_VAR


//Fill output data
IF b_enableMonitor THEN
	Output.w_Status.0	:=	Monitor.ACswitchgear.b_OutputMCCBfb;
	Output.w_Status.1	:=	Monitor.ACswitchgear.b_PENlinkfb;
	//Output.w_Status.2	:=	Monitor.ACswitchgear.?.b_GridConStatus;
	
	Output.w_Warnings.0	:=	Monitor.ACswitchgear.b_CEEprefuseOK;
	Output.w_Warnings.1	:=	Monitor.ACswitchgear.b_OutputMCCBShuntOK;
	Output.w_Warnings.2	:=	Monitor.powermonitor.events.b_MBCommWarning OR Monitor.powermonitor.events.b_MBTimeoutWarning;
	Output.w_Warnings.3	:=	Monitor.protections.OvercurrentProtection.b_OutputWarning;
	
	Output.w_Faults.0	:=	Monitor.protections.OvercurrentProtection.b_OutputAlarm;
	Output.w_Faults.1	:=	Monitor.powermonitor.events.b_MBCommError;

	Output.i_ActivePower 			:=	RealToint (	In	:= Monitor.powermonitor.OutputField.r_ActivePower, 	Scale	:=	10);
	Output.i_ReactivePower 			:=	RealToint (	In	:= Monitor.powermonitor.OutputField.r_ReactivePower, Scale	:=	10);
	Output.ui_frequency				:=	RealToUint(	In	:= Monitor.powermonitor.OutputField.r_Frequency, 	Scale	:=	10);
	Output.ui_VoltageL1N			:=	RealToUint(	In	:= Monitor.powermonitor.OutputField.r_PhaseVoltage[1], Scale	:=	10);
	Output.ui_VoltageL2N			:=	RealToUint(	In	:= Monitor.powermonitor.OutputField.r_PhaseVoltage[2], Scale	:=	10);
	Output.ui_VoltageL3N			:=	RealToUint(	In	:= Monitor.powermonitor.OutputField.r_PhaseVoltage[3], Scale	:=	10);
	Output.ui_VoltageL1L2			:=	RealToUint(	In	:= Monitor.powermonitor.OutputField.r_LineVoltage[1], Scale	:=	10);
	Output.ui_VoltageL2L3			:=	RealToUint(	In	:= Monitor.powermonitor.OutputField.r_LineVoltage[2], Scale	:=	10);
	Output.ui_VoltageL3L1			:=	RealToUint(	In	:= Monitor.powermonitor.OutputField.r_LineVoltage[3], Scale	:=	10);
	Output.i_CurrentL1				:=	RealToint (	In	:= Monitor.powermonitor.OutputField.r_Current[1], 	Scale	:=	10);
	Output.i_CurrentL2				:=	RealToint (	In	:= Monitor.powermonitor.OutputField.r_Current[2], 	Scale	:=	10);
	Output.i_CurrentL3				:=	RealToint (	In	:= Monitor.powermonitor.OutputField.r_Current[3], 	Scale	:=	10);
	Output.i_CurrentN				:=	RealToint (	In	:= Monitor.powermonitor.OutputField.r_Current[4], 	Scale	:=	10);
	
	Output.ui_TotalEnergyConsumed_high	:= UDINT_TO_UINT(SHR(RealToUdint(	In	:=	monitor.powermonitor.OutputField.r_EnergyConsumed, Scale	:=	10), 16));
	Output.ui_TotalEnergyConsumed_low	:= UDINT_TO_UINT(RealToUdint(	In	:=	monitor.powermonitor.OutputField.r_EnergyConsumed, Scale	:=	10));
	Output.ui_TotalEnergySupplied_high 	:= UDINT_TO_UINT(SHR(RealToUdint(	In	:=	monitor.powermonitor.OutputField.r_EnergySupplied, Scale	:=	10), 16));
	Output.ui_TotalEnergySupplied_low 	:= UDINT_TO_UINT(RealToUdint(	In	:=	monitor.powermonitor.OutputField.r_EnergySupplied, Scale	:=	10));
END_IF
END_METHOD

METHOD MapPeakShaveBox : BOOL
VAR_INPUT
	Input	:	ST_PNInput_PeakShaveBox;
END_VAR

VAR_OUTPUT
	Output	:	ST_PNOutput_PeakShaveBox;
END_VAR
	
//Fill output data
IF b_enableMonitor THEN
	Output.w_Status.0	:=	Monitor.peakshavebox.Buscoupler.b_SlaveReady;

	Output.w_Warnings.0	:=	Monitor.peakshavebox.Powermonitor.StatusWord.b_Warning;
	Output.w_Warnings.1	:=	Monitor.peakshavebox.Powermonitor.StatusWord.b_Over_1 OR	
							Monitor.peakshavebox.Powermonitor.StatusWord.b_Over_2 OR	
							Monitor.peakshavebox.Powermonitor.StatusWord.b_Over_3 OR	
							Monitor.peakshavebox.Powermonitor.StatusWord.b_Over_4;	

	Output.w_Faults.0	:=	Monitor.peakshavebox.Powermonitor.StatusWord.b_Error;

	Output.i_ActivePower 		:=	RealToint (	In	:= 	Monitor.peakshavebox.Powermonitor.Data.r_ActivePowerL1 + 
														Monitor.peakshavebox.Powermonitor.Data.r_ActivePowerL2 +
														Monitor.peakshavebox.Powermonitor.Data.r_ActivePowerL3 , 	scale := 10);
														
	Output.i_ReactivePower 		:=	RealToint(	In	:= 	Monitor.peakshavebox.Powermonitor.Data.r_ReactivePowerL1 + 
														Monitor.peakshavebox.Powermonitor.Data.r_ReactivePowerL2 +
														Monitor.peakshavebox.Powermonitor.Data.r_ReactivePowerL3 , 	scale := 10);
														
	Output.ui_frequency			:=	RealToUint(	In	:= Monitor.peakshavebox.Powermonitor.Data.r_FrequencyL1, 		Scale	:=	10);
	Output.ui_VoltageL1N		:=	RealToUint(	In	:= Monitor.peakshavebox.Powermonitor.Data.r_VoltageL1N_RMS, 	Scale	:=	10);
	Output.ui_VoltageL2N		:=	RealToUint(	In	:= Monitor.peakshavebox.Powermonitor.Data.r_VoltageL2N_RMS, 	Scale	:=	10);
	Output.ui_VoltageL3N		:=	RealToUint(	In	:= Monitor.peakshavebox.Powermonitor.Data.r_VoltageL3N_RMS, 	Scale	:=	10);
	Output.ui_VoltageL1L2		:=	RealToUint(	In	:= Monitor.peakshavebox.Powermonitor.Data.r_VoltageL1L2_RMS, 	Scale	:=	10);
	Output.ui_VoltageL2L3		:=	RealToUint(	In	:= Monitor.peakshavebox.Powermonitor.Data.r_VoltageL2L3_RMS, 	Scale	:=	10);
	Output.ui_VoltageL3L1		:=	RealToUint(	In	:= Monitor.peakshavebox.Powermonitor.Data.r_VoltageL3L1_RMS, 	Scale	:=	10);
	Output.i_CurrentL1			:=	RealToint (	In	:= Monitor.peakshavebox.Powermonitor.Data.r_CurrentL1_RMS, 		Scale	:=	10);
	Output.i_CurrentL2			:=	RealToint (	In	:= Monitor.peakshavebox.Powermonitor.Data.r_CurrentL2_RMS, 		Scale	:=	10);
	Output.i_CurrentL3			:=	RealToint (	In	:= Monitor.peakshavebox.Powermonitor.Data.r_CurrentL3_RMS, 		Scale	:=	10);
	Output.i_CurrentN			:=	RealToint (	In	:= Monitor.peakshavebox.Powermonitor.Data.r_CurrentN_RMS, 		Scale	:=	10);
END_IF

//process input data
IF NOT get.events.b_HeartBeatLost AND b_enableControl THEN
	Input.w_ControlBits;	//not in use
	SoftSettings.PSB.setpointTimeslot1.r_FeedInCurrentLimitSoft	:=	UintToReal(in	:= Input.ui_FeedInCurrentLimit, Scale := 10);
	SoftSettings.PSB.setpointTimeslot1.r_SupplyCurrentLimitSoft	:=	UintToReal(in	:= Input.ui_SupplyCurrentLimit, Scale := 10);
	SoftSettings.PSB.setpointTimeslot1.r_IdleChargePower		:=	UintToReal(in	:= Input.UI_IdleChargePower, Scale := 10);
	SoftSettings.PSB.setpointTimeslot1.r_SocTarget				:=	UintToReal(in	:= Input.UI_SOCTarget, Scale := 10);
END_IF
END_METHOD

METHOD MapPowerSTack : BOOL
VAR_INPUT
	Input	:	ST_PNInput_PowerStack;
END_VAR

VAR_OUTPUT
	Output	:	ST_PNOutput_Powerstack;
END_VAR

//Fill output data
IF b_enableMonitor THEN
	Output.w_Status.0	:=	Monitor.powerstack.Netcontactor.b_NetConFb;
	Output.w_Status.1	:=	Monitor.powerstack.b_ACDetected;
	Output.w_Status.2	:=	Monitor.powerstack.b_DCDetected;
	Output.w_Status.3	:=	Monitor.powerstack.b_InverterRunning;
	Output.w_Status.4	:=	Monitor.powerstack.b_ControlEnabled;

	Output.w_Warnings.0	:=	Monitor.powerstack.Events.b_MasterWarning;
	Output.w_Warnings.1	:=	Monitor.powerstack.Events.b_SlaveWarning;
	
	Output.w_Faults.0	:=	Monitor.powerstack.Events.b_MasterFault;
	Output.w_Faults.1	:=	Monitor.powerstack.Events.b_SlaveFault;
	Output.w_Faults.2	:=	Monitor.powerstack.Events.b_NetcontactorFault;
	
	Output.w_PowerStackStatus 	:= Monitor.powerstack.e_Status;
	Output.w_InverterMode		:= Monitor.powerstack.e_InverterMode;
	Output.w_Powermode			:= Monitor.powerstack.e_PowerMode;	
	
	Output.i_ActivePower				:=  RealToint 	(	In	:= Monitor.powerstack.r_ActivePower, 	Scale	:=	10);
	Output.i_ReactivePower 				:= 	RealToint 	(	In	:= Monitor.powerstack.r_ReactivePower, 	Scale	:=	10);
	Output.ui_D7_Voltage				:=  RealToUint 	(	In	:= Monitor.powerstack.r_ACVoltageD7, 	Scale	:=	10);
	Output.ui_D7_frequency 				:=  RealToUint	(	In	:= Monitor.powerstack.r_FrequencyD7, 	Scale	:=	10);
	Output.i_ACCurrent					:=  RealToint 	(	In	:= Monitor.powerstack.r_AcCurrent, 		Scale	:=	10);
	Output.i_ActivePowerSetpoint 		:=  RealToint 	(	In	:= Operation.system.r_Pset, 			Scale	:=	10);
	Output.i_ReactivePowerSetpoint 		:=  RealToint 	(	In	:= Operation.system.r_Qset, 			Scale	:=	10);
	Output.ui_PFSetpoint				:=  RealToUint	( 	In	:= Operation.system.r_PFset, 			Scale	:=	10);
	Output.ui_LoadPercentage			:=	RealToUint 	( 	IN 	:= Monitor.powerstack.r_LoadPercent, 	Scale	:=	10);
	Output.ui_RatedCurrent				:=	RealToUint	( 	In	:= Monitor.powerstack.r_RatedCurrent, 	Scale	:=	10);
	Output.ui_RatedPower				:=	RealToUint	( 	In	:= Monitor.powerstack.r_RatedPower, 	Scale	:=	10);
END_IF

//process input data
IF NOT get.events.b_HeartBeatLost AND b_enableControl THEN
	Operation.system.b_PFsetEnable 				:=	Input.w_ControlBits.0;	
	Operation.system.b_NetContactorForceClose 	:=	Input.w_ControlBits.1;	
	Operation.system.b_NetContactorSyncClose 	:=	Input.w_ControlBits.2;	
	
	CASE Input.w_GridMode OF
		0:	SoftSettings.system.e_Gridmode := eGridMode.auto;
		1:	SoftSettings.system.e_Gridmode := eGridMode.following;
		2:	SoftSettings.system.e_Gridmode := eGridMode.forming;
	END_CASE
	
	CASE Input.w_PowerMode OF
		0:	SoftSettings.system.e_PowerMode := ePowerMode.auto;
		1:	SoftSettings.system.e_PowerMode := ePowerMode.FixedPower;
		2:	SoftSettings.system.e_PowerMode := ePowerMode.Droop;
		3:	SoftSettings.system.e_PowerMode := ePowerMode.DroopZeroStart;
	END_CASE

	Operation.system.r_NominalVoltage	:=	UintToReal(in:= Input.ui_NominalVoltage, scale := 10);
	Operation.system.r_NominalFrequency	:=	UintToReal(in:= Input.ui_NominalFrequency, scale := 10);
	Operation.system.r_Pset				:=	IntToReal(in:= Input.i_Pset, scale := 10);
	Operation.system.r_Qset	 			:=	IntToReal(in:= Input.i_Qset, scale := 10);
	Operation.system.r_PFset 			:=	UintToReal(in:= Input.ui_PFset, scale := 10);
	Softsettings.system.r_FrequencyDroop	:=	UintToReal(in:= Input.ui_FrequencyDroop, scale := 10);
	Softsettings.system.r_VoltageDroop		:=	UintToReal(in:= Input.ui_VoltageDroop, scale := 10);
	SoftSettings.system.r_Pmax				:=	UintToReal(in:= Input.ui_Pmax, scale := 10);
	SoftSettings.system.r_Pmin				:=	UintToReal(in:= Input.ui_Pmin, scale := 10);
	SoftSettings.system.r_Qmax				:=	UintToReal(in:= Input.ui_Qmax, scale := 10);
	SoftSettings.system.r_Qmin				:=	UintToReal(in:= Input.ui_Qmin, scale := 10);
	//SoftSettings.system.ACCurrentLimit		:=	UintToReal(in:= Input.ui_ACCurrentLimit, scale := 10);
	//SoftSettings.system.ApparentPowerLimit	:=	UintToReal(in:= Input.ui_ApparentPowerLimit, scale := 10);
	SoftSettings.system.r_PowerRampRate 	:= UintToReal(in:= Input.ui_PowerRampRate, scale := 10);
ELSE
	//If Heartbeat fails or control is not allowed --> reset Operational values
	// soft settings may remain.
	Operation.system.r_Pset	 :=	0;
	Operation.system.r_Qset	 :=	0;
	Operation.system.r_PFset :=	1;
END_IF
END_METHOD

METHOD MapZPT : BOOL
VAR_OUTPUT
	Output	:	ST_PNOutput_ZPT;
END_VAR

VAR
	HighestTemp	:	Real;
END_VAR


//Fill output data
IF b_enableMonitor THEN
	Output.w_Status;	//not in use
	
	Output.w_Warnings.0	:=	Monitor.neutraltransformer.events.b_OvercurrentWarning;
	Output.w_Warnings.1	:=	Monitor.neutraltransformer.events.b_TemperatureHighPhase[1] OR 
							Monitor.neutraltransformer.events.b_TemperatureHighPhase[2] OR 
							Monitor.neutraltransformer.events.b_TemperatureHighPhase[3];
	Output.w_Warnings.2	:=	Monitor.neutraltransformer.events.b_VoltageUnbalanceHigh;
	Output.w_Warnings.3	:=	Monitor.neutraltransformer.events.b_NeutralCurrentHigh;
	
	Output.w_Faults.0	:=	Monitor.neutraltransformer.events.b_OvercurrentAlarm;
	Output.w_Faults.1	:=	Monitor.neutraltransformer.events.b_TemperatureTooHighPhase[1] OR 
							Monitor.neutraltransformer.events.b_TemperatureTooHighPhase[2] OR 
							Monitor.neutraltransformer.events.b_TemperatureTooHighPhase[3];
	Output.w_Faults.2	:=	Monitor.neutraltransformer.events.b_VoltageUnbalanceTooHigh;
	Output.w_Faults.3	:=	Monitor.neutraltransformer.events.b_NeutralCurrentTooHigh;

	Output.ui_RatedPower:=	0; //where to find?
	Output.ui_PowerLoad	:=	RealToUint(in:=Monitor.neutraltransformer.r_Powerload, Scale:=10);
	
	HighestTemp := MAX(Monitor.neutraltransformer.r_TemperaturePhase[0], Monitor.neutraltransformer.r_TemperaturePhase[1], Monitor.neutraltransformer.r_TemperaturePhase[2]);
	Output.i_TransformerTemperature	:=	RealToint(in:=HighestTemp, Scale:=10);

END_IF
END_METHOD

METHOD PNCouplerDiagnostics : BOOL
VAR_INPUT
	DevState	:	WORD;
	DevDiag		:	WORD;
END_VAR
Get.events.b_DeviceFault 				:= FALSE;
get.events.b_NetworkConfigurationFault 	:= FALSE;
get.events.b_NetworkConfigurationFault 	:= FALSE;
get.events.b_DataConfigurationFault 	:= FALSE;

CASE DevState OF
	0:
		IF Get.events.b_HeartBeatLost THEN
			Get.eControllerStatus := e_ControllerStatus.Ready;
		ELSE
			Get.eControllerStatus := e_ControllerStatus.Active;
		END_IF
	1:
		Get.eControllerStatus := e_ControllerStatus.Init;
	2,7,8,9:
		Get.eControllerStatus := e_ControllerStatus.Error;
		Get.events.b_DeviceFault := TRUE;
	3,4,5,6,10,11,12:		
		Get.events.b_DeviceFault := TRUE;
		get.events.b_NetworkConfigurationFault := TRUE;
	13,14,15,16:
		Get.events.b_DeviceFault := TRUE;
		get.events.b_DataConfigurationFault := TRUE;
END_CASE
END_METHOD

METHOD RealToInt : INT
VAR_INPUT
	In		:	REAL;
	Scale	:	UINT := 10;
END_VAR
RealToInt := REAL_TO_INT(LIMIT(-32768, In*Scale, 32767));
END_METHOD

METHOD RealToUDINT : UDINT
VAR_INPUT
	In		:	REAL;
	Scale	:	UINT := 10;
END_VAR
RealToUdint := REAL_TO_UDINT(LIMIT(0, In*Scale, 4294967295));
END_METHOD

METHOD RealToUint : UINT
VAR_INPUT
	In		:	REAL;
	Scale	:	UINT := 10;
END_VAR
RealToUint := REAL_TO_UINT(LIMIT(0, In*Scale, 65535));
END_METHOD

METHOD Reset : BOOL
VAR_INPUT
END_VAR

//?

Reset := True;
END_METHOD

METHOD UintToReal : REAL
VAR_INPUT
	in		:	UINT;
	Scale	:	UINT := 10;
END_VAR
UintToReal := UINT_TO_REAL(in)/Scale;
END_METHOD

END_FUNCTION_BLOCK

// ---- POUs/Objects/BMS/FB_BMS.TcPOU
FUNCTION_BLOCK FB_BMS
VAR_OUTPUT
	PowerStatus: eHVDC_Powerstatus := 0;
END_VAR
VAR_INPUT
	Set : st_BMS_Set;
END_VAR

VAR_OUTPUT
	BMSGet: st_BMS_GetStatus;
END_VAR

VAR	
	FBState				:	ePOUState;
	IO					:	FB_BMS_IO;
	HWControl			:	st_BMS_IO;
	
	InitTimeout			: 	TON := (PT:=T#3S);
	
	BMS_230V_StartupTimer : TON := (PT := TIME#3S0MS);
	BMS_24V_StartupTimer : TON := (PT := TIME#2S0MS);
	
	TempVar				: WORD;
	SFCInit				: BOOL := FALSE;
	SFCReset			: BOOL := FALSE;
	
//	by_CommErrorCounter	:	BYTE	:=	0;
	b_MBComErrorActive	: 	BOOL 	:= FALSE;
	
	ResetBMS	:	Bool; 
	b_BMSShutdownRequested: BOOL;
	
	BMSReadIntervalTimer	 : TON := (PT := TIME#1S0MS);
END_VAR

(*
FB_BMS

Inputs
	Set.b_EnableBMS				:	BOOL;
		Start BMS SFC sequence and initializes BMS. False means full BMS powerdown, so no status logging.
		With HVDC enabled, setting this value to False has no effect. Only after HVDC powerdown this value is tested.
		
	Set.b_ClearFault				:	BOOL;
		Clear errors and warning in BMS system. Set to true to initiate reset. Value resets automatically to false.
	
	Set.b_HVDC_Required			: 	BOOL;
		Set by FB_internalPowersupply. True initiates and keeps HVDC on, False initiates and retains powerdown

Outputs
	BMSGET
		-Some general status info
		-BATTinfo	struct with main operation battery data
		-MBMU_Status 	struct with detailed MBMU data
		-SBMU			Struct with detailed data per SBMU
		-Events			Warnings & Errors as per Sunspec list.
*)

IO(HWControl:=HWControl);

BMSReadIntervalTimer(in:= not BMSReadIntervalTimer.Q);

//Reset ErrorActive before entering SFC. 
//any remaining error in the Modbus methods will set Erroractive again. 
//This is pushed to events in BMS_Diagnostics

//TEMPBMSHB();
//hv required not allowed if BMS not enabled
set.b_HVDC_Required := set.b_HVDC_Required AND Set.b_EnableBMS;
//shutdown allowed if hvdc is offline
b_BMSShutdownRequested := (NOT Set.b_EnableBMS) AND BMSGet.BattInfo.ui_BMS_PowerOnStatus <> ePowerOnStatus.On; 

//b_MBComErrorActive := FALSE;

IF FBState = ePOUState.EMSTOP THEN
	Set.b_HVDC_Required := FALSE;
END_IF

BMSSFC();


IF ResetBMS THEN
	Reset();
END_IF


BMS_Diagnostics();

ACTION aBMSPoweroff:
HWControl.b_BMS_230V_Enable := FALSE;
HWControl.b_BMS_24V_Enable := FALSE;

BMSGet.BattInfo.b_BMSHeartBeatOK := FALSE;
BMSGet.BattInfo.ui_BMS_PowerOnStatus := ePowerOnStatus.Off;
BMSGet.BattInfo.ui_BMS_Status := eBMS_Status.Off;

BMSGet.MBMU_Status.BatteryStatus.b_BMSHeartBeatOK := FALSE;
BMSGet.MBMU_Status.BatteryStatus.ui_BMS_PowerOnStatus := ePowerOnStatus.Off;
BMSGet.MBMU_Status.BatteryStatus.ui_BMS_Status := eBMS_Status.Off;

FBState := ePOUState.OFF;
END_ACTION

ACTION aBMSPowerOn:

//230V inverter requires some startup time. Start this first to init SBMU before MBMU
//This may not be needed, but the idea is to make sure the MBMU can reach the SBMU's at boot.
FBState := ePOUState.PowerUp;
HWControl.b_BMS_230V_Enable := TRUE;
BMS_230V_StartupTimer(IN:=HWControl.b_BMS_230V_Enable);

HWControl.b_BMS_24V_Enable := BMS_230V_StartupTimer.Q;
BMS_24V_StartupTimer(IN:=HWControl.b_BMS_24V_Enable);
END_ACTION

ACTION aClearFaults:
SFCTip := ClearBMSFaults();
END_ACTION

ACTION aDisableInsulationMonitor:
SFCTip := OpenInsulationSwitch(TRUE);
END_ACTION

ACTION aGetMBMUData:
SFCTip := GetMBMUData();
END_ACTION

ACTION aGetSBMUData:
SFCTip := GetSBMUData();
END_ACTION

ACTION aGetStaticData:

IF (TempVar=0) THEN
	IF GetMBMUStaticSystemData() THEN
		TempVar:=1;
	END_IF;
ELSE
	IF GetSBMUStaticSystemData(TempVar) THEN
		TempVar := TempVar+1;
	END_IF
	
	IF TempVar > 4 then//BMSGet.MBMU_Status.by_NumberOfSubSystems THEN
		TempVar:=0;
		SFCTip := TRUE;
	END_IF
END_IF
END_ACTION

ACTION aGetStatus:
IF GetSystemStatus() THEN
	IF FBState = ePOUState.PowerUp THEN FBState := ePOUState.Init; END_IF
	SFCTip := TRUE;
END_IF
END_ACTION

ACTION aInit:
TempVar := 0;
SFCReset := false;
END_ACTION

ACTION aSetDateTime:
SFCTip := SetBMSDateTime();
END_ACTION

ACTION aSetPowerMode:
SFCTip := SetPowerMode();
END_ACTION

ACTION aWatchdog:
IF FBState = ePOUState.Init THEN FBState := ePOUState.Normal; END_IF

SFCTip := BMSHeartBeat();
TempVar := 0;
END_ACTION

METHOD BMS_Diagnostics : BOOL
VAR
	
END_VAR

BMSGet.Events.b_COMMUNICATION_ERROR				:=	BMSGet.MBMU_Status.GeneralSBMUStatus[6].5 	//SBMU CCAN comm lost
												OR BMSGet.MBMU_Status.GeneralSBMUStatus[6].6 	//SBMU SCAN comm lost
												OR BMSGet.MBMU_Status.GeneralSBMUStatus[6].7	//SBMU MCAN comm lost
												OR BMSGet.MBMU_Status.MBMUStatus[0].6			//MBMU MCAN comm warning
												OR BMSGet.MBMU_Status.MBMUStatus[0].7			//MBMU MCAN comm Lost
												OR BMSGet.MBMU_Status.MBMUStatus[0].8			//SBMU EMS COMM lost
												OR BMSGet.MBMU_Status.MBMUStatus[3].4			//SBMU MBMU comm fault
												OR b_MBComErrorActive;					//One or more Modbus communication errors 
									
BMSGet.Events.b_OVER_TEMP_ALARM					:= BMSGet.MBMU_Status.GeneralSBMUStatus[2].1;	//single cell Overtemperature warning 4

BMSGet.Events.b_OVER_TEMP_WARNING				:= BMSGet.MBMU_Status.GeneralSBMUStatus[1].14	//single cell Overtemperature warning 1
												OR BMSGet.MBMU_Status.GeneralSBMUStatus[2].0; 	//single cell Overtemperature warning 2

BMSGet.Events.b_UNDER_TEMP_ALARM				:= FALSE; //no data

BMSGet.Events.b_UNDER_TEMP_WARNING				:= BMSGet.MBMU_Status.GeneralSBMUStatus[2].2	//single cell Undertemperature warning 1
												OR BMSGet.MBMU_Status.GeneralSBMUStatus[2].3 	//single cell Undertemperature warning 2
												OR BMSGet.MBMU_Status.GeneralSBMUStatus[2].4; 	//single cell Undertemperature warning 3

BMSGet.Events.b_OVER_CHARGE_CURRENT_ALARM		:= BMSGet.MBMU_Status.GeneralSBMUStatus[1].9;	//Charge Overcurrent warning 4

BMSGet.Events.b_OVER_CHARGE_CURRENT_WARNING		:= BMSGet.MBMU_Status.GeneralSBMUStatus[1].6	//Charge Overcurrent warning 1
												OR BMSGet.MBMU_Status.GeneralSBMUStatus[1].7 	//Charge Overcurrent warning 2
												OR BMSGet.MBMU_Status.GeneralSBMUStatus[1].8; 	//Charge Overcurrent warning 3
											
BMSGet.Events.b_OVER_DISCHARGE_CURRENT_ALARM	:= BMSGet.MBMU_Status.GeneralSBMUStatus[1].5;	//Discharge Overcurrent warning 4

BMSGet.Events.b_OVER_DISCHARGE_CURRENT_WARNING	:= BMSGet.MBMU_Status.GeneralSBMUStatus[1].2	//Discharge Overcurrent warning 1
												OR BMSGet.MBMU_Status.GeneralSBMUStatus[1].3 	//Discharge Overcurrent warning 2
												OR BMSGet.MBMU_Status.GeneralSBMUStatus[1].4; 	//Discharge Overcurrent warning 3
											
BMSGet.Events.b_OVER_VOLT_ALARM					:= BMSGet.MBMU_Status.GeneralSBMUStatus[0].6;	//Single cell extreme overVoltage warning

BMSGet.Events.b_OVER_VOLT_WARNING				:= BMSGet.MBMU_Status.GeneralSBMUStatus[0].0	//Single cell overVoltage warning 1
												OR BMSGet.MBMU_Status.GeneralSBMUStatus[0].1 	//Single cell overVoltage warning 2
												OR BMSGet.MBMU_Status.GeneralSBMUStatus[0].2 	//Single cell overVoltage warning 3
												OR BMSGet.MBMU_Status.GeneralSBMUStatus[0].8 	//Single rack overVoltage warning 1
												OR BMSGet.MBMU_Status.GeneralSBMUStatus[0].9; 	//Single rack overVoltage warning 2
												
BMSGet.Events.b_UNDER_VOLT_ALARM				:= BMSGet.MBMU_Status.GeneralSBMUStatus[0].7;	//Single cell extreme underVoltage warning

BMSGet.Events.b_UNDER_VOLT_WARNING				:= BMSGet.MBMU_Status.GeneralSBMUStatus[0].3	//Single cell underVoltage warning 1
												OR BMSGet.MBMU_Status.GeneralSBMUStatus[0].4 	//Single cell underVoltage warning 2
												OR BMSGet.MBMU_Status.GeneralSBMUStatus[0].5 	//Single cell underVoltage warning 3
												OR BMSGet.MBMU_Status.GeneralSBMUStatus[0].10 	//Single rack underVoltage warning 1
												OR BMSGet.MBMU_Status.GeneralSBMUStatus[0].11; //Single rack underVoltage warning 2
												
BMSGet.Events.b_UNDER_SOC_MIN_ALARM				:= BMSGet.MBMU_Status.GeneralSBMUStatus[6].14;	//r_SOC low warning 2

BMSGet.Events.b_UNDER_SOC_MIN_WARNING			:= BMSGet.MBMU_Status.GeneralSBMUStatus[6].13;	//r_SOC low warning 1

BMSGet.Events.b_OVER_SOC_MAX_ALARM				:= FALSE; //no data

BMSGet.Events.b_OVER_SOC_MAX_WARNING			:= FALSE; //no data

BMSGet.Events.b_VOLTAGE_IMBALANCE_WARNING		:= BMSGet.MBMU_Status.GeneralSBMUStatus[0].12;	//large voltage difference warning

BMSGet.Events.b_TEMPERATURE_IMBALANCE_ALARM		:= FALSE; //no data
												
BMSGet.Events.b_TEMPERATURE_IMBALANCE_WARNING	:= BMSGet.MBMU_Status.GeneralSBMUStatus[2].5	//Large temperature difference warning 1
												OR BMSGet.MBMU_Status.GeneralSBMUStatus[2].6 	//Large temperature difference warning 2
												OR BMSGet.MBMU_Status.GeneralSBMUStatus[2].7; 	//Large temperature difference warning 3
												
BMSGet.Events.b_CONTACTOR_ERROR					:= BMSGet.MBMU_Status.GeneralSBMUStatus[5].1	//Main positive relay sticking
												OR BMSGet.MBMU_Status.GeneralSBMUStatus[5].2 	//Main negative relay sticking
												OR BMSGet.MBMU_Status.GeneralSBMUStatus[5].3 	//Both main relays sticking
												OR BMSGet.MBMU_Status.GeneralSBMUStatus[5].4 	//Main positive relay open
												OR BMSGet.MBMU_Status.GeneralSBMUStatus[5].5 	//Main negative relay open
												OR BMSGet.MBMU_Status.GeneralSBMUStatus[6].15; //HV open circuit warning
												
BMSGet.Events.b_FAN_ERROR						:= BMSGet.MBMU_Status.GeneralSBMUStatus[5].7;	//main control box fan warning

BMSGet.Events.b_GROUND_FAULT					:= FALSE; //no data

BMSGet.Events.b_OPEN_DOOR_ERROR					:= FALSE; //no data

BMSGet.Events.b_CURRENT_IMBALANCE_WARNING		:= FALSE; //no data

BMSGet.Events.b_OTHER_ALARM						:= BMSGet.MBMU_Status.GeneralSBMUStatus[0].13	//Invalid voltage warning
												OR BMSGet.MBMU_Status.GeneralSBMUStatus[1].10 	//Current sensor fault
												OR BMSGet.MBMU_Status.GeneralSBMUStatus[2].15 //single temperature sampling abnormal value warning
												OR BMSGet.MBMU_Status.GeneralSBMUStatus[3].0 	//multiple temperature sampling abnormal value warning
												OR BMSGet.MBMU_Status.GeneralSBMUStatus[4].9 	//CSC supply abnormal
												OR BMSGet.MBMU_Status.GeneralSBMUStatus[4].10 	//SBMU supply abnormal
												OR BMSGet.MBMU_Status.GeneralSBMUStatus[4].14 	//MSD warning
												OR BMSGet.MBMU_Status.GeneralSBMUStatus[4].15 	//rack fuse warning
												OR BMSGet.MBMU_Status.GeneralSBMUStatus[6].11 	//cell balance circuit short
												OR BMSGet.MBMU_Status.GeneralSBMUStatus[7].3 	//precharching failed twice
												OR BMSGet.MBMU_Status.MBMUStatus[1].7 			//estop fault
												OR BMSGet.MBMU_Status.MBMUStatus[3].3; 		//MBMU 24V fault
												
BMSGet.Events.b_OTHER_WARNING					:= BMSGet.MBMU_Status.MBMUStatus[0].0 			//insulation warning
												OR BMSGet.MBMU_Status.MBMUStatus[1].10 		//rack fan warning
												OR BMSGet.MBMU_Status.MBMUStatus[3].7;			//TMS warning
												
BMSGet.Events.b_CONFIGURATION_ALARM				:= BMSGet.MBMU_Status.GeneralSBMUStatus[5].0	//rack isolate switch warning
												OR BMSGet.MBMU_Status.GeneralSBMUStatus[5].6 	//battery rack door fault
												OR BMSGet.MBMU_Status.GeneralSBMUStatus[5].9 	//rack fire system level 1 fault
												OR BMSGet.MBMU_Status.GeneralSBMUStatus[5].10 	//smoke detector contact open
												OR BMSGet.MBMU_Status.GeneralSBMUStatus[5].11 	//temp detector contact open
												OR BMSGet.MBMU_Status.GeneralSBMUStatus[5].14 	//aerosol warning
												OR BMSGet.MBMU_Status.GeneralSBMUStatus[6].0 	//rack fire system level 2 fault
												OR BMSGet.MBMU_Status.GeneralSBMUStatus[6].10 	//SBMU TMS CCAN comm lost with hv on
												OR BMSGet.MBMU_Status.GeneralSBMUStatus[7].0 	//lvl 3 fault tms
												OR BMSGet.MBMU_Status.GeneralSBMUStatus[7].1 	//TMS mode conflict
												OR BMSGet.MBMU_Status.GeneralSBMUStatus[7].2 	//TMS warning
												OR BMSGet.MBMU_Status.GeneralSBMUStatus[8].0 	//Thermal runaway caused fire
												OR BMSGet.MBMU_Status.MBMUStatus[0].1	 		//Insulation fault
												OR BMSGet.MBMU_Status.MBMUStatus[0].2			//Insulation error
												OR BMSGet.MBMU_Status.MBMUStatus[0].3 			//Less HV racks than expected
												OR BMSGet.MBMU_Status.MBMUStatus[0].9			//IMM comm fault
												OR BMSGet.MBMU_Status.MBMUStatus[0].10 		//Air conditioning comm fault
												OR BMSGet.MBMU_Status.MBMUStatus[0].11			//TMS comm fault
												OR BMSGet.MBMU_Status.MBMUStatus[0].13			//TMS comm fault lvl 2
												OR BMSGet.MBMU_Status.MBMUStatus[0].14 		//TMS mode conflict
												OR BMSGet.MBMU_Status.MBMUStatus[0].15			//TMS comm fault level 1
												OR BMSGet.MBMU_Status.MBMUStatus[1].3	 		//AUX power DCDC failure
												OR BMSGet.MBMU_Status.MBMUStatus[1].4			//Fire system fault lvl 1
												OR BMSGet.MBMU_Status.MBMUStatus[1].5 			//Fire system fault lvl 2
												OR BMSGet.MBMU_Status.MBMUStatus[1].6			//Fire system failure warning
												OR BMSGet.MBMU_Status.MBMUStatus[1].8	 		//client estop fault
												OR BMSGet.MBMU_Status.MBMUStatus[1].9			//rack door fault
												OR BMSGet.MBMU_Status.MBMUStatus[1].12;		//smoke ex fan body fault
								
BMSGet.Events.b_CONFIGURATION_WARNING			:= BMSGet.MBMU_Status.GeneralSBMUStatus[6].8	//SBMU TMS CCAN comm lost
												OR BMSGet.MBMU_Status.MBMUStatus[0].12	 		//TMS comm warning
												OR BMSGet.MBMU_Status.MBMUStatus[1].0			//SPD failure
												OR BMSGet.MBMU_Status.MBMUStatus[1].1 			//Aux power DCDC failure
												OR BMSGet.MBMU_Status.MBMUStatus[1].2			//AUX power DCDC failure
												OR BMSGet.MBMU_Status.MBMUStatus[1].6 			//Fire system failure warning
												OR BMSGet.MBMU_Status.MBMUStatus[1].11;		//Smoke exhaust fan body warning
END_METHOD

METHOD BMSHeartBeat : BOOL

VAR_INST
	WriteReg		:	FB_MBWriteSingleReg;
	ReadReg			:	FB_MBReadRegs;
	
	readbCommBusy		:	BOOL;
	readbComError		:	BOOL;
	readerrID			:	UDINT;
	
	WritebCommBusy		:	BOOL;
	WritebComError		:	BOOL;
	WriteerrID			:	UDINT;
	
	ReadDone			:	F_Trig;
	ReadOK				: 	BOOL;
	WriteDone			:	F_Trig;
	WriteOK				: 	BOOL;
	
	ComTimer		:	Ton := (PT := TIME#0S200MS);
	
	OldValue		:	WORD := 0;
	BMSHBValue		:	WORD := 0;
	
	WatchdogUpdateTimer	:	Tof := (PT := TIME#3S0MS);
	WatchdogCommTimer	:	Tof := (PT := TIME#3S0MS);
	
	ComRetryCounter	:	USINT := 0;
END_VAR

ComTimer(in := NOT(ComTimer.Q));

ReadReg(
sIPAddr := Config.IP_BMS,
nTCPPort := Config.MBPort_BMS,
nUnitID := 255,//16#FF;
nMBAddr := 768,
nQuantity := 1,
cbLength := 2,
pDestAddr := ADR(BMSHBValue),
bExecute := ComTimer.Q,
tTimeout := T#100MS,
bBusy => readbCommBusy,
bError => readbComError,
nErrId => readerrID,
cbRead => 
);

ReadDone(clk := readbCommBusy);
ReadOK := ReadDone.Q AND NOT readbComError;


//read value is transmitted back into the write buffer if read is succesful
//BMS increments this value every second.
WriteReg(
sIPAddr := Config.IP_BMS,
nTCPPort := Config.MBPort_BMS,
nUnitID := 255,//16#FF;
nMBAddr := 896,
nValue := BMSHBValue,
tTimeout := T#100MS,
bExecute := ReadOK,
bBusy => WritebCommBusy,
bError => WritebComError,
nErrId => WriteerrID,
);

WriteDone(clk := writebCommBusy);
WriteOK := writeDone.Q AND NOT writebComError;

//if written value and BMS value are equal for longer than 3 seconds, the BMS isn't incrementing the value anymore or communication failed.
//BMS itself will throw warning after 30s and disable 10s after that.
WatchdogUpdateTimer(in:= (OldValue <> BMSHBValue));
OldValue := BMSHBValue;

//if modbus communication throws an error retry for 3s, otherwise system failed.
//WatchdogCommTimer(in:= WriteOK);

//both values are normally high and fall away if they timeout
BMSGet.BattInfo.b_BMSHeartBeatOK := WatchdogUpdateTimer.Q;// OR WatchdogCommTimer.Q;
BMSGet.MBMU_Status.BatteryStatus.b_BMSHeartBeatOK := WatchdogUpdateTimer.Q;

IF (ReadDone.Q AND readbComError) OR (WriteDone.Q AND WritebComError) THEN
	ComRetryCounter := ComRetryCounter + 1;
	IF COMRetryCounter > 5 THEN
		b_MBComErrorActive := TRUE;
		BMSGet.BattInfo.b_BMSHeartBeatOK := FALSE;
	END_IF
END_IF

IF WriteOK THEN
	ComRetryCounter := 0;
	BMSHeartBeat := TRUE;
END_IF
END_METHOD

ACTION BMSSFC:
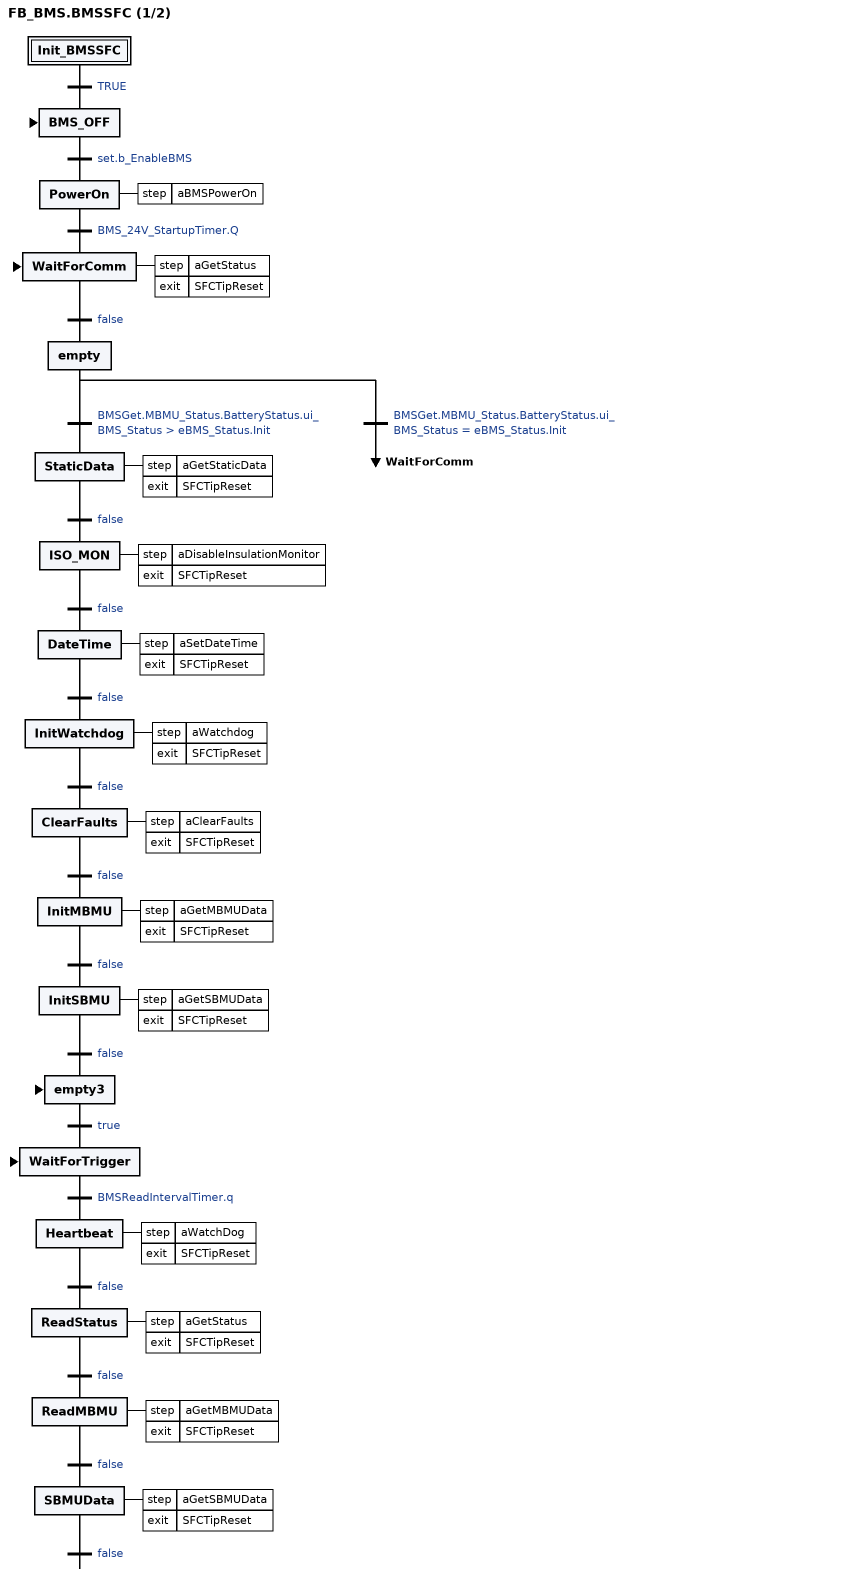
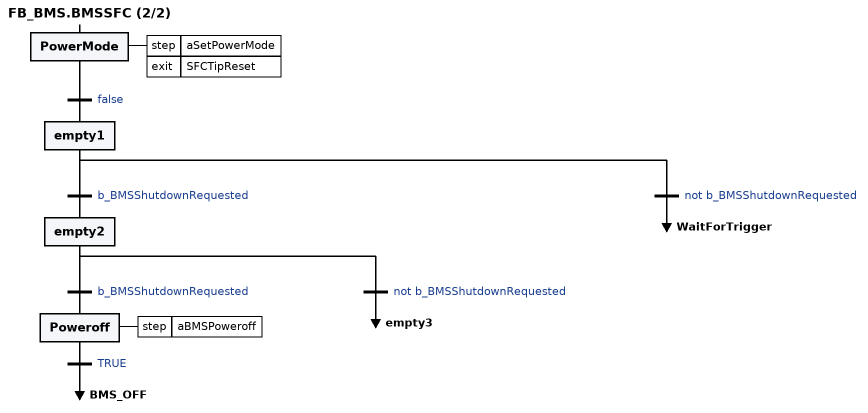
INITIAL_STEP Init_BMSSFC:
END_STEP
TRANSITION FROM Init_BMSSFC TO BMS_OFF
    := TRUE;
END_TRANSITION
STEP BMS_OFF:
END_STEP
TRANSITION FROM BMS_OFF TO PowerOn
    := set.b_EnableBMS;
END_TRANSITION
// macro BMSInit begins
STEP PowerOn:
    aBMSPowerOn(N);  // step action
END_STEP
TRANSITION FROM PowerOn TO WaitForComm
    := BMS_24V_StartupTimer.Q;
END_TRANSITION
STEP WaitForComm:
    aGetStatus(N);  // step action
    SFCTipReset(P0);  // exit action
END_STEP
TRANSITION FROM WaitForComm TO empty
    := false;
END_TRANSITION
STEP empty:
END_STEP
TRANSITION FROM empty TO StaticData
    := BMSGet.MBMU_Status.BatteryStatus.ui_BMS_Status > eBMS_Status.Init;
END_TRANSITION
TRANSITION FROM empty TO WaitForComm
    := BMSGet.MBMU_Status.BatteryStatus.ui_BMS_Status = eBMS_Status.Init;
END_TRANSITION
STEP StaticData:
    aGetStaticData(N);  // step action
    SFCTipReset(P0);  // exit action
END_STEP
TRANSITION FROM StaticData TO ISO_MON
    := false;
END_TRANSITION
STEP ISO_MON:
    aDisableInsulationMonitor(N);  // step action
    SFCTipReset(P0);  // exit action
END_STEP
TRANSITION FROM ISO_MON TO DateTime
    := false;
END_TRANSITION
STEP DateTime:
    aSetDateTime(N);  // step action
    SFCTipReset(P0);  // exit action
END_STEP
TRANSITION FROM DateTime TO InitWatchdog
    := false;
END_TRANSITION
STEP InitWatchdog:
    aWatchdog(N);  // step action
    SFCTipReset(P0);  // exit action
END_STEP
TRANSITION FROM InitWatchdog TO ClearFaults
    := false;
END_TRANSITION
STEP ClearFaults:
    aClearFaults(N);  // step action
    SFCTipReset(P0);  // exit action
END_STEP
TRANSITION FROM ClearFaults TO InitMBMU
    := false;
END_TRANSITION
STEP InitMBMU:
    aGetMBMUData(N);  // step action
    SFCTipReset(P0);  // exit action
END_STEP
TRANSITION FROM InitMBMU TO InitSBMU
    := false;
END_TRANSITION
STEP InitSBMU:
    aGetSBMUData(N);  // step action
    SFCTipReset(P0);  // exit action
END_STEP
TRANSITION FROM InitSBMU TO empty3
    := false;
END_TRANSITION
STEP empty3:
END_STEP
TRANSITION FROM empty3 TO WaitForTrigger
    := true;
END_TRANSITION
// macro BMSActive begins
STEP WaitForTrigger:
END_STEP
TRANSITION FROM WaitForTrigger TO Heartbeat
    := BMSReadIntervalTimer.q;
END_TRANSITION
STEP Heartbeat:
    aWatchDog(N);  // step action
    SFCTipReset(P0);  // exit action
END_STEP
TRANSITION FROM Heartbeat TO ReadStatus
    := false;
END_TRANSITION
STEP ReadStatus:
    aGetStatus(N);  // step action
    SFCTipReset(P0);  // exit action
END_STEP
TRANSITION FROM ReadStatus TO ReadMBMU
    := false;
END_TRANSITION
STEP ReadMBMU:
    aGetMBMUData(N);  // step action
    SFCTipReset(P0);  // exit action
END_STEP
TRANSITION FROM ReadMBMU TO SBMUData
    := false;
END_TRANSITION
STEP SBMUData:
    aGetSBMUData(N);  // step action
    SFCTipReset(P0);  // exit action
END_STEP
TRANSITION FROM SBMUData TO PowerMode
    := false;
END_TRANSITION
STEP PowerMode:
    aSetPowerMode(N);  // step action
    SFCTipReset(P0);  // exit action
END_STEP
TRANSITION FROM PowerMode TO empty1
    := false;
END_TRANSITION
STEP empty1:
END_STEP
TRANSITION FROM empty1 TO empty2
    := b_BMSShutdownRequested;
END_TRANSITION
TRANSITION FROM empty1 TO WaitForTrigger
    := not b_BMSShutdownRequested;
END_TRANSITION
STEP empty2:
END_STEP
TRANSITION FROM empty2 TO Poweroff
    := b_BMSShutdownRequested;
END_TRANSITION
TRANSITION FROM empty2 TO empty3
    := not b_BMSShutdownRequested;
END_TRANSITION
STEP Poweroff:
    aBMSPoweroff(N);  // step action
END_STEP
TRANSITION FROM Poweroff TO BMS_OFF
    := TRUE;
END_TRANSITION
// branch label Branch1_BMSSFC
// branch label Branch0_BMSSFC
END_ACTION

METHOD ClearBMSFaults : BOOL
VAR_INST
	WriteRegSet		:	FB_MBWriteSingleReg;
	WriteRegClear	:	FB_MBWriteSingleReg;
	ComTimer	:	Ton := (PT := TIME#200MS);
	
	bCommBusy	:	BOOL;
	bComError	:	BOOL;
	errID		:	UDINT;
	b_ClearDone	:	BOOL := FALSE;

	w_ClearFault	:	WORD;
	TX1Done 	: 	f_trig;
	
	bCommBusy2	:	BOOL;
	bComError2	:	BOOL;
	errID2		:	UDINT;
	TX2Done 	: 	f_trig;

	ComRetryCounter	:	USINT := 0;	
END_VAR
//Catl says we need to write 1 to clear, then write back to 0 to be able to log new errors.
//This method is called continuously when bms is active. It will usually write zero's.
//If set.b_ClearFault is 1, that will be written. The value will be cleared by this method after the write so next write will be a 0 again.
//With this, a reset cycle takes half a second with the current ComTimer.

ClearBMSFaults := FALSE;

ComTimer(in := NOT(ComTimer.Q));

//first write clearing register to 1
WriteRegSet(
	sIPAddr := Config.IP_BMS,
	nTCPPort := Config.MBPort_BMS,
	nUnitID := 255,//16#FF;
	nMBAddr := 908,
	nValue := 1,
	tTimeout := T#100MS,
	bExecute := ComTimer.Q,
	bBusy => bCommBusy,
	bError => bComError,
	nErrId => errID,
);

TX1Done(CLK := bCommBusy);
b_ClearDone	:= 	TX1Done.Q AND NOT bComError;

//reset value back to 0 afterwards. CATL requirement
WriteRegClear(
	sIPAddr := Config.IP_BMS,
	nTCPPort := Config.MBPort_BMS,
	nUnitID := 255,//16#FF;
	nMBAddr := 908,
	nValue := 0,
	tTimeout := T#100MS,
	bExecute := b_ClearDone,
	bBusy => bCommBusy2,
	bError => bComError2,
	nErrId => errID2
);

TX2Done(CLK := bCommBusy2);

IF (TX1Done.Q AND bComError) OR (TX2Done.Q AND bComError2) THEN
	ComRetryCounter := ComRetryCounter + 1;
	IF COMRetryCounter > 5 THEN
		b_MBComErrorActive := TRUE;
	END_IF
END_IF

IF TX2Done.Q AND NOT bComError2 THEN
	ComRetryCounter := 0;
	ClearBMSFaults := TRUE;
END_IF
END_METHOD

METHOD EMSTOP : BOOL
VAR_INPUT
	EMSTOP_Active	:	BOOL;
END_VAR
EMSTOP := FALSE;

FBState := ePOUState.EMSTOP;
set.b_HVDC_Required := FALSE;

IF BMSGet.BattInfo.ui_BMS_PowerOnStatus = ePowerOnStatus.Off THEN
	EMSTOP := TRUE;
END_IF
END_METHOD

METHOD GetCellData : BOOL
VAR_INPUT
	SBMUID	:	BYTE;	//SBMU 1-#ofstrings
	CSCID	:	BYTE;	//CSC 1-4
END_VAR

VAR_OUTPUT
	CellVoltages		:	ARRAY[1..52] OF REAL;
	Celltemperatures	:	ARRAY[1..16] OF INT;
	BalanceStatus		:	ARRAY[1..4] OF WORD; //bit per cell?
END_VAR

VAR_INST
	MBReadCellVoltages	: 	FB_MBReadRegs;
	MBReadTemperatures	: 	FB_MBReadRegs;
	MBReadCellBalance	: 	FB_MBReadRegs;
	
//	CellVoltageData		: 	ARRAY[1..52] OF WORD;
	TemperatureData		: 	ARRAY[1..16] OF BYTE;
//	CellBalanceData		: 	ARRAY[1..4] OF WORD;
	
	bCommBusy			:	ARRAY[1..3] OF BOOL;
	bComError			:	ARRAY[1..3] OF BOOL;
	errID				:	ARRAY[1..3] OF UDINT;
	cbRead				:	ARRAY[1..3] OF UDINT;
	TransmissionDone	: 	ARRAY[1..3] OF f_trig;
	
	DataComplete		:	ARRAY[1..3] OF BOOL;
	
	ComTimer			:	Ton := (PT := TIME#0S500MS);
END_VAR

VAR
	LoopCounter			:	INT;
END_VAR

GetCellData := FALSE;

IF (SBMUID < 1) OR (SBMUID > BMSGet.MBMU_Status.by_NumberOfSubSystems) THEN
	GetCellData := TRUE;
	RETURN;
END_IF
IF (CSCID < 1) OR (CSCID > 4) THEN
	GetCellData := TRUE;
	RETURN;
END_IF

ComTimer(in := NOT(ComTimer.Q));

IF ComTimer.Q THEN
	DataComplete[1] := FALSE;
	DataComplete[2] := FALSE;
	DataComplete[3] := FALSE;
END_IF

MBReadCellVoltages(
sIPAddr := Config.IP_BMS,
nTCPPort := Config.MBPort_BMS,
nUnitID := 255,//16#FF;
nMBAddr := (SBMUID*1024)+128+(52*(CSCID-1)),	//SBMU 1, module 1, start at 0x0480, increment 52 per module & 1024 per sbmu
nQuantity := 52,
cbLength := SIZEOF(CellVoltages),
pDestAddr := ADR(CellVoltages),
bExecute := ComTimer.Q,
bBusy => bCommBusy[1],
bError => bComError[1],
nErrId => errID[1],
cbRead => cbRead[1]
);

MBReadTemperatures(
sIPAddr := Config.IP_BMS,
nTCPPort := Config.MBPort_BMS,
nUnitID := 1,//16#FF;
nMBAddr := (SBMUID*1024)+704+(8*(CSCID-1)),	//SBMU 1, module 1, start at 0x06c0, increment 8 (16 byte) per module & 1024 per sbmu
nQuantity := 8*2,
cbLength := SIZEOF(TemperatureData),
pDestAddr := ADR(TemperatureData),
bExecute := ComTimer.Q,
bBusy => bCommBusy[2],
bError => bComError[2],
nErrId => errID[2],
cbRead => cbRead[2]
);

MBReadTemperatures(
sIPAddr := Config.IP_BMS,
nTCPPort := Config.MBPort_BMS,
nUnitID := 1,//16#FF;
nMBAddr := (SBMUID*1024)+912+(4*(CSCID-1)),	//SBMU 1, module 1, start at 0x0790, increment 4 per module & 1024 per sbmu
											//not sure if CSC2 starts at address 4, or immediatly follows after last cell of csc1.
nQuantity := 4*2,
cbLength := SIZEOF(BalanceStatus),
pDestAddr := ADR(BalanceStatus),
bExecute := ComTimer.Q,
bBusy => bCommBusy[3],
bError => bComError[3],
nErrId => errID[3],
cbRead => cbRead[3]
);

TransmissionDone[1](clk:=bCommBusy[1]);
TransmissionDone[2](clk:=bCommBusy[2]);
TransmissionDone[3](clk:=bCommBusy[3]);

IF TransmissionDone[1].Q AND NOT bComError[1] THEN
	DataComplete[1] := TRUE;
END_IF

IF TransmissionDone[2].Q AND NOT bComError[2] THEN
	FOR loopcounter := 1 TO 16 BY 1 DO
		Celltemperatures[loopcounter] := TemperatureData[loopcounter]-50;
	END_FOR
	DataComplete[2] := TRUE;
END_IF

IF TransmissionDone[1].Q AND NOT bComError[1] THEN
	DataComplete[3] := TRUE;
END_IF

GetCellData := DataComplete[1] AND DataComplete[2] AND DataComplete[3];
END_METHOD

METHOD GetDiagnostics 
VAR_IN_OUT
	AddError		: ARRAY [*] OF FB_AddErrorST;
	a_ActiveEvents	: ARRAY [*] OF ST_ErrorStruct;
	w_Index			: WORD;
END_VAR

VAR_OUTPUT
	b_errorActive	: BOOL;
	b_warningActive	: BOOL;
END_VAR

VAR
	by_errCt	: BYTE;
	by_warnCt	: BYTE;
	w_ID		: WORD;
END_VAR
(*BMS errors (sunspec)*)
	(*BMS Communication error*)		AddError[w_Index](
			in_b_ErrorTrig			:= BMSGet.Events.b_COMMUNICATION_ERROR,
			out_ST_Error			:= a_ActiveEvents[w_Index],
			w_ID					:= 1 + w_ID,
			s_Message				:= 'BMS communication error',
			e_sev					:= eSeverity.EmergencyShutdown,	//<-- maybe normal shutdown?
			in_b_AutoClear			:= FALSE,
			in_t_TriggerTime		:= TIME#1000MS,
			//in_e_ErrAckAccess		:= TRUE,
			);
		IF AddError[w_Index].b_out THEN by_errCt := by_errCt + 1; END_IF;
		w_Index := w_Index +1;
		
	(*Configuration fault*)		AddError[w_Index](
			in_b_ErrorTrig			:= BMSGet.Events.b_CONFIGURATION_ALARM,
			out_ST_Error			:= a_ActiveEvents[w_Index],
			w_ID					:= 1 + w_ID,
			s_Message				:= 'BMS configuration error',
			e_sev					:= eSeverity.NormalShutdown,
			in_b_AutoClear			:= FALSE,
			//in_t_TriggerTime		:= TIME#500MS,
			//in_e_ErrAckAccess		:= TRUE,
			);
		IF AddError[w_Index].b_out THEN by_errCt := by_errCt + 1; END_IF;
		w_Index := w_Index +1;
	
	(*Configuration warning*)		AddError[w_Index](
			in_b_ErrorTrig			:= BMSGet.Events.b_CONFIGURATION_WARNING,
			out_ST_Error			:= a_ActiveEvents[w_Index],
			w_ID					:= 1 + w_ID,
			s_Message				:= 'BMS configuration error',
			e_sev					:= eSeverity.Warning,
			in_b_AutoClear			:= FALSE,
			//in_t_TriggerTime		:= TIME#500MS,
			//in_e_ErrAckAccess		:= TRUE,
			);
		IF AddError[w_Index].b_out THEN by_errCt := by_errCt + 1; END_IF;
		w_Index := w_Index +1;
		
	(*Contactor fault*)		AddError[w_Index](
			in_b_ErrorTrig			:= BMSGet.Events.b_CONTACTOR_ERROR,
			out_ST_Error			:= a_ActiveEvents[w_Index],
			w_ID					:= 1 + w_ID,
			s_Message				:= 'BMS Contactor fault',
			e_sev					:= eSeverity.EmergencyShutdown,
			in_b_AutoClear			:= FALSE,
			//in_t_TriggerTime		:= TIME#500MS,
			//in_e_ErrAckAccess		:= TRUE,
			);
		IF AddError[w_Index].b_out THEN by_errCt := by_errCt + 1; END_IF;
		w_Index := w_Index +1;
		
	(*Current imbalance warning*)		AddError[w_Index](						//unused, will always be false
			in_b_ErrorTrig			:= BMSGet.Events.b_CURRENT_IMBALANCE_WARNING,
			out_ST_Error			:= a_ActiveEvents[w_Index],
			w_ID					:= 1 + w_ID,
			s_Message				:= 'BMS Current imbalance warning',
			e_sev					:= eSeverity.Warning,
			in_b_AutoClear			:= FALSE,
			//in_t_TriggerTime		:= TIME#500MS,
			//in_e_ErrAckAccess		:= TRUE,
			);
		IF AddError[w_Index].b_out THEN by_errCt := by_errCt + 1; END_IF;
		w_Index := w_Index +1;
		
	(*Fan error*)		AddError[w_Index](
			in_b_ErrorTrig			:= BMSGet.Events.b_FAN_ERROR,
			out_ST_Error			:= a_ActiveEvents[w_Index],
			w_ID					:= 1 + w_ID,
			s_Message				:= 'BMS fan error',
			e_sev					:= eSeverity.NormalShutdown,
			in_b_AutoClear			:= FALSE,
			//in_t_TriggerTime		:= TIME#500MS,
			//in_e_ErrAckAccess		:= TRUE,
			);
		IF AddError[w_Index].b_out THEN by_errCt := by_errCt + 1; END_IF;
		w_Index := w_Index +1;

	(*Ground fault*)		AddError[w_Index](
			in_b_ErrorTrig			:= BMSGet.Events.b_GROUND_FAULT,		//unused, will always be false
			out_ST_Error			:= a_ActiveEvents[w_Index],
			w_ID					:= 1 + w_ID,
			s_Message				:= 'BMS Insulation fault',
			e_sev					:= eSeverity.EmergencyShutdown,
			in_b_AutoClear			:= FALSE,
			//in_t_TriggerTime		:= TIME#500MS,
			//in_e_ErrAckAccess		:= TRUE,
			);
		IF AddError[w_Index].b_out THEN by_errCt := by_errCt + 1; END_IF;
		w_Index := w_Index +1;

	(*Door open error*)		AddError[w_Index](							//unused, will always be false
			in_b_ErrorTrig			:= BMSGet.Events.b_OPEN_DOOR_ERROR,
			out_ST_Error			:= a_ActiveEvents[w_Index],
			w_ID					:= 1 + w_ID,
			s_Message				:= 'BMS door open',
			e_sev					:= eSeverity.NormalShutdown,
			in_b_AutoClear			:= FALSE,
			//in_t_TriggerTime		:= TIME#500MS,
			//in_e_ErrAckAccess		:= TRUE,
			);
		IF AddError[w_Index].b_out THEN by_errCt := by_errCt + 1; END_IF;
		w_Index := w_Index +1;

	(*misc alarm*)		AddError[w_Index](							
			in_b_ErrorTrig			:= BMSGet.Events.b_OTHER_ALARM,
			out_ST_Error			:= a_ActiveEvents[w_Index],
			w_ID					:= 1 + w_ID,
			s_Message				:= 'BMS miscellaneous error',
			e_sev					:= eSeverity.NormalShutdown,
			in_b_AutoClear			:= FALSE,
			//in_t_TriggerTime		:= TIME#500MS,
			//in_e_ErrAckAccess		:= TRUE,
			);
		IF AddError[w_Index].b_out THEN by_errCt := by_errCt + 1; END_IF;
		w_Index := w_Index +1;
		
	(*misc warning*)		AddError[w_Index](							
			in_b_ErrorTrig			:= BMSGet.Events.b_OTHER_WARNING,
			out_ST_Error			:= a_ActiveEvents[w_Index],
			w_ID					:= 1 + w_ID,
			s_Message				:= 'BMS miscellaneous warning',
			e_sev					:= eSeverity.Warning,
			in_b_AutoClear			:= FALSE,
			//in_t_TriggerTime		:= TIME#500MS,
			//in_e_ErrAckAccess		:= TRUE,
			);
		IF AddError[w_Index].b_out THEN by_errCt := by_errCt + 1; END_IF;
		w_Index := w_Index +1;

	(*Overcharge current alarm*)		AddError[w_Index](							
			in_b_ErrorTrig			:= BMSGet.Events.b_OVER_CHARGE_CURRENT_ALARM,
			out_ST_Error			:= a_ActiveEvents[w_Index],
			w_ID					:= 1 + w_ID,
			s_Message				:= 'BMS Charge current too high error',
			e_sev					:= eSeverity.NormalShutdown,			
			in_b_AutoClear			:= FALSE,									
			//in_t_TriggerTime		:= TIME#500MS,
			//in_e_ErrAckAccess		:= TRUE,
			);
		IF AddError[w_Index].b_out THEN by_errCt := by_errCt + 1; END_IF;
		w_Index := w_Index +1;
		
	(*Overcharge current warning*)		AddError[w_Index](							
			in_b_ErrorTrig			:= BMSGet.Events.b_OVER_CHARGE_CURRENT_WARNING,
			out_ST_Error			:= a_ActiveEvents[w_Index],
			w_ID					:= 1 + w_ID,
			s_Message				:= 'BMS Charge current too high warning',
			e_sev					:= eSeverity.Warning,				//<-- Powerstack should lower the power
			in_b_AutoClear			:= FALSE,								
			//in_t_TriggerTime		:= TIME#500MS,
			//in_e_ErrAckAccess		:= TRUE,
			);
		IF AddError[w_Index].b_out THEN by_errCt := by_errCt + 1; END_IF;
		w_Index := w_Index +1;
		
	(*OverDischarge current Alarm*)		AddError[w_Index](							
			in_b_ErrorTrig			:= BMSGet.Events.b_OVER_DISCHARGE_CURRENT_ALARM,
			out_ST_Error			:= a_ActiveEvents[w_Index],
			w_ID					:= 1 + w_ID,
			s_Message				:= 'BMS Discharge current too high error',
			e_sev					:= eSeverity.NormalShutdown,				
			in_b_AutoClear			:= FALSE,								
			//in_t_TriggerTime		:= TIME#500MS,
			//in_e_ErrAckAccess		:= TRUE,
			);
			
		IF AddError[w_Index].b_out THEN by_errCt := by_errCt + 1; END_IF;
		w_Index := w_Index +1;
		
	(*OverDischarge current warning*)		AddError[w_Index](							
			in_b_ErrorTrig			:= BMSGet.Events.b_OVER_DISCHARGE_CURRENT_WARNING,
			out_ST_Error			:= a_ActiveEvents[w_Index],
			w_ID					:= 1 + w_ID,
			s_Message				:= 'BMS Discharge current too high warning',
			e_sev					:= eSeverity.Warning,				//<-- Powerstack should lower the power
			in_b_AutoClear			:= FALSE,								
			//in_t_TriggerTime		:= TIME#500MS,
			//in_e_ErrAckAccess		:= TRUE,
			);
		IF AddError[w_Index].b_out THEN by_errCt := by_errCt + 1; END_IF;
		w_Index := w_Index +1;
		
	(*Overcharge r_SOC error*)		AddError[w_Index](							//unused, will remain false
			in_b_ErrorTrig			:= BMSGet.Events.b_OVER_SOC_MAX_ALARM,
			out_ST_Error			:= a_ActiveEvents[w_Index],
			w_ID					:= 1 + w_ID,
			s_Message				:= 'BMS r_SOC too high error',
			e_sev					:= eSeverity.NormalShutdown,				
			in_b_AutoClear			:= FALSE,								
			//in_t_TriggerTime		:= TIME#500MS,
			//in_e_ErrAckAccess		:= TRUE,
			);
		IF AddError[w_Index].b_out THEN by_errCt := by_errCt + 1; END_IF;
		w_Index := w_Index +1;
		
	(*Overcharge r_SOC error*)		AddError[w_Index](							//unused, will remain false
			in_b_ErrorTrig			:= BMSGet.Events.b_OVER_SOC_MAX_WARNING,
			out_ST_Error			:= a_ActiveEvents[w_Index],
			w_ID					:= 1 + w_ID,
			s_Message				:= 'BMS r_SOC too high warning',
			e_sev					:= eSeverity.Warning,				
			in_b_AutoClear			:= FALSE,								
			//in_t_TriggerTime		:= TIME#500MS,
			//in_e_ErrAckAccess		:= TRUE,
			);
		IF AddError[w_Index].b_out THEN by_errCt := by_errCt + 1; END_IF;
		w_Index := w_Index +1;
		
	(*OverDischarge r_SOC error*)		AddError[w_Index](							
			in_b_ErrorTrig			:= BMSGet.Events.b_UNDER_SOC_MIN_ALARM,
			out_ST_Error			:= a_ActiveEvents[w_Index],
			w_ID					:= 1 + w_ID,
			s_Message				:= 'BMS r_SOC too low error',
			e_sev					:= eSeverity.NormalShutdown,				
			in_b_AutoClear			:= FALSE,								
			//in_t_TriggerTime		:= TIME#500MS,
			//in_e_ErrAckAccess		:= TRUE,
			);
		IF AddError[w_Index].b_out THEN by_errCt := by_errCt + 1; END_IF;
		w_Index := w_Index +1;
		
	(*OverDischarge r_SOC error*)		AddError[w_Index](							
			in_b_ErrorTrig			:= BMSGet.Events.b_UNDER_SOC_MIN_WARNING,
			out_ST_Error			:= a_ActiveEvents[w_Index],
			w_ID					:= 1 + w_ID,
			s_Message				:= 'BMS r_SOC too low warning',
			e_sev					:= eSeverity.Warning,				
			in_b_AutoClear			:= FALSE,								
			//in_t_TriggerTime		:= TIME#500MS,
			//in_e_ErrAckAccess		:= TRUE,
			);
		IF AddError[w_Index].b_out THEN by_errCt := by_errCt + 1; END_IF;
		w_Index := w_Index +1;
		
	(*OverTemperature error*)		AddError[w_Index](							
			in_b_ErrorTrig			:= BMSGet.Events.b_OVER_TEMP_ALARM,
			out_ST_Error			:= a_ActiveEvents[w_Index],
			w_ID					:= 1 + w_ID,
			s_Message				:= 'Battery Overtemperature error',
			e_sev					:= eSeverity.NormalShutdown,				
			in_b_AutoClear			:= FALSE,								
			//in_t_TriggerTime		:= TIME#500MS,
			//in_e_ErrAckAccess		:= TRUE,
			);
		IF AddError[w_Index].b_out THEN by_errCt := by_errCt + 1; END_IF;
		w_Index := w_Index +1;		

	(*OverTemperature warning*)		AddError[w_Index](							
			in_b_ErrorTrig			:= BMSGet.Events.b_OVER_TEMP_WARNING,
			out_ST_Error			:= a_ActiveEvents[w_Index],
			w_ID					:= 1 + w_ID,
			s_Message				:= 'Battery Overtemperature warning',
			e_sev					:= eSeverity.Warning,				
			in_b_AutoClear			:= FALSE,								
			//in_t_TriggerTime		:= TIME#500MS,
			//in_e_ErrAckAccess		:= TRUE,
			);
		IF AddError[w_Index].b_out THEN by_errCt := by_errCt + 1; END_IF;
		w_Index := w_Index +1;
	
	(*OverVoltage error*)		AddError[w_Index](							
			in_b_ErrorTrig			:= BMSGet.Events.b_OVER_VOLT_ALARM,
			out_ST_Error			:= a_ActiveEvents[w_Index],
			w_ID					:= 1 + w_ID,
			s_Message				:= 'Battery overvoltage error',
			e_sev					:= eSeverity.NormalShutdown,				
			in_b_AutoClear			:= FALSE,								
			//in_t_TriggerTime		:= TIME#500MS,
			//in_e_ErrAckAccess		:= TRUE,
			);
		IF AddError[w_Index].b_out THEN by_errCt := by_errCt + 1; END_IF;
		w_Index := w_Index +1;		

	(*OverVoltage warning*)		AddError[w_Index](							
			in_b_ErrorTrig			:= BMSGet.Events.b_OVER_VOLT_WARNING,
			out_ST_Error			:= a_ActiveEvents[w_Index],
			w_ID					:= 1 + w_ID,
			s_Message				:= 'Battery overvoltage warning',
			e_sev					:= eSeverity.Warning,				
			in_b_AutoClear			:= FALSE,								
			//in_t_TriggerTime		:= TIME#500MS,
			//in_e_ErrAckAccess		:= TRUE,
			);
		IF AddError[w_Index].b_out THEN by_errCt := by_errCt + 1; END_IF;
		w_Index := w_Index +1;
		
	(*Temperature imbalance error*)		AddError[w_Index](							
			in_b_ErrorTrig			:= BMSGet.Events.b_TEMPERATURE_IMBALANCE_ALARM,
			out_ST_Error			:= a_ActiveEvents[w_Index],
			w_ID					:= 1 + w_ID,
			s_Message				:= 'Battery temperature imbalance error',
			e_sev					:= eSeverity.NormalShutdown,				
			in_b_AutoClear			:= FALSE,								
			//in_t_TriggerTime		:= TIME#500MS,
			//in_e_ErrAckAccess		:= TRUE,
			);
		IF AddError[w_Index].b_out THEN by_errCt := by_errCt + 1; END_IF;
		w_Index := w_Index +1;		

	(*Temperature imbalance warning*)		AddError[w_Index](							
			in_b_ErrorTrig			:= BMSGet.Events.b_TEMPERATURE_IMBALANCE_WARNING,
			out_ST_Error			:= a_ActiveEvents[w_Index],
			w_ID					:= 1 + w_ID,
			s_Message				:= 'Battery temperature imbalance warning',
			e_sev					:= eSeverity.Warning,				
			in_b_AutoClear			:= FALSE,								
			//in_t_TriggerTime		:= TIME#500MS,
			//in_e_ErrAckAccess		:= TRUE,
			);
		IF AddError[w_Index].b_out THEN by_errCt := by_errCt + 1; END_IF;
		w_Index := w_Index +1;

	(*Under Temperature error*)		AddError[w_Index](							
			in_b_ErrorTrig			:= BMSGet.Events.b_UNDER_TEMP_ALARM,
			out_ST_Error			:= a_ActiveEvents[w_Index],
			w_ID					:= 1 + w_ID,
			s_Message				:= 'Battery temperature low error',
			e_sev					:= eSeverity.NormalShutdown,				
			in_b_AutoClear			:= FALSE,								
			//in_t_TriggerTime		:= TIME#500MS,
			//in_e_ErrAckAccess		:= TRUE,
			);
		IF AddError[w_Index].b_out THEN by_errCt := by_errCt + 1; END_IF;
		w_Index := w_Index +1;		

	(*Under Temperature warning*)		AddError[w_Index](							
			in_b_ErrorTrig			:= BMSGet.Events.b_UNDER_TEMP_WARNING,
			out_ST_Error			:= a_ActiveEvents[w_Index],
			w_ID					:= 1 + w_ID,
			s_Message				:= 'Battery temperature low warning',
			e_sev					:= eSeverity.Warning,				
			in_b_AutoClear			:= FALSE,								
			//in_t_TriggerTime		:= TIME#500MS,
			//in_e_ErrAckAccess		:= TRUE,
			);
		IF AddError[w_Index].b_out THEN by_errCt := by_errCt + 1; END_IF;
		w_Index := w_Index +1;

	(*Under Temperature error*)		AddError[w_Index](							
			in_b_ErrorTrig			:= BMSGet.Events.b_UNDER_VOLT_ALARM,
			out_ST_Error			:= a_ActiveEvents[w_Index],
			w_ID					:= 1 + w_ID,
			s_Message				:= 'Battery undervoltage error',
			e_sev					:= eSeverity.NormalShutdown,				
			in_b_AutoClear			:= FALSE,								
			//in_t_TriggerTime		:= TIME#500MS,
			//in_e_ErrAckAccess		:= TRUE,
			);
		IF AddError[w_Index].b_out THEN by_errCt := by_errCt + 1; END_IF;
		w_Index := w_Index +1;		

	(*Under Temperature warning*)		AddError[w_Index](							
			in_b_ErrorTrig			:= BMSGet.Events.b_UNDER_VOLT_WARNING,
			out_ST_Error			:= a_ActiveEvents[w_Index],
			w_ID					:= 1 + w_ID,
			s_Message				:= 'Battery undervoltage warning',
			e_sev					:= eSeverity.Warning,				
			in_b_AutoClear			:= FALSE,								
			//in_t_TriggerTime		:= TIME#500MS,
			//in_e_ErrAckAccess		:= TRUE,
			);
		IF AddError[w_Index].b_out THEN by_errCt := by_errCt + 1; END_IF;
		w_Index := w_Index +1;
		
	(*Battery voltage imbalance warning*)		AddError[w_Index](							
			in_b_ErrorTrig			:= BMSGet.Events.b_VOLTAGE_IMBALANCE_WARNING,
			out_ST_Error			:= a_ActiveEvents[w_Index],
			w_ID					:= 1 + w_ID,
			s_Message				:= 'Battery voltage imbalance warning',
			e_sev					:= eSeverity.Warning,				
			in_b_AutoClear			:= FALSE,								
			//in_t_TriggerTime		:= TIME#500MS,
			//in_e_ErrAckAccess		:= TRUE,
			);
		IF AddError[w_Index].b_out THEN by_errCt := by_errCt + 1; END_IF;
		w_Index := w_Index +1;
END_METHOD

METHOD GetMBMUData : BOOL
VAR_INST
	
	MBReadMBMU			: 	FB_MBReadRegs;
	MBMUData 			: 	ARRAY[0..52] OF WORD;
	bCommBusy			:	BOOL;
	bComError			:	BOOL;
	errID				:	UDINT;
	cbRead				:	UDINT;
	TransmissionDone	: 	f_trig;
	COMretryCounter		:	USINT := 0;
	
	ComTimer			:	Ton := (PT := TIME#0S200MS);
END_VAR

VAR
	Counter				:	INT;
END_VAR
//read mbmu data every 100ms

GetMBMUData := FALSE;

ComTimer(in := NOT(ComTimer.Q));

MBReadMBMU(
sIPAddr := Config.IP_BMS,
nTCPPort := Config.MBPort_BMS,
nUnitID := 255,//16#FF;
nMBAddr := 0,
nQuantity := 53,
cbLength := SIZEOF(MBMUData),
pDestAddr := ADR(MBMUData),
bExecute := ComTimer.Q,
bBusy => bCommBusy,
bError => bComError,
nErrId => errID,
cbRead => cbRead,
tTimeout := T#100MS
);

TransmissionDone(CLK := bCommBusy);

IF TransmissionDone.Q THEN
	IF NOT bComError THEN
		MEMCPY(ADR(BMSGet.MBMU_Status.GeneralSBMUStatus[0]), ADR(MBMUData[0]), 32);	//0x0000 - 0x000f
		MEMCPY(ADR(BMSGet.MBMU_Status.MBMUStatus[0]), ADR(MBMUData[16]), 32);			//0x0010 - 0x001f
	
		BMSGet.MBMU_Status.BatteryStatus.r_SystemVoltage := WORD_TO_REAL(MBMUData[32])/10; 						//0-1500V with 0.1V/bit
		BMSGet.MBMU_Status.BatteryStatus.r_SystemCurrent := WORD_TO_REAL(MBMUData[33])-20000; 					//-20k .. +20k kW in 1kW/bit steps
		
		BMSGet.MBMU_Status.BatteryStatus.r_SOC := WORD_TO_REAL(MBMUData[34])/10; 								//0-100% with 0.1%/bit;
		BMSGet.MBMU_Status.BatteryStatus.r_SOH := WORD_TO_REAL(MBMUData[35])/10; 								//0-100% with 0.1%/bit;
		
		BMSGet.MBMU_Status.BatteryStatus.CellVoltage[eSubValues.Maximum] := WORD_TO_REAL(MBMUData[36])/1000;	//0-5v with 0.001v/bit;
		BMSGet.MBMU_Status.BatteryStatus.CellVoltage[eSubValues.Minimum] := WORD_TO_REAL(MBMUData[37])/1000;	//0-5v with 0.001v/bit;
		BMSGet.MBMU_Status.BatteryStatus.CellVoltage[eSubValues.Average] := WORD_TO_REAL(MBMUData[38])/1000;	//0-5v with 0.001v/bit;
		
		BMSGet.MBMU_Status.BatteryStatus.CellTemperature[eSubValues.Maximum] := WORD_TO_REAL(MBMUData[39])-50;	//-50..200gr with 1gr/bit;
		BMSGet.MBMU_Status.BatteryStatus.CellTemperature[eSubValues.Minimum] := WORD_TO_REAL(MBMUData[40])-50;	//-50..200gr with 1gr/bit;
		BMSGet.MBMU_Status.BatteryStatus.CellTemperature[eSubValues.Average] := WORD_TO_REAL(MBMUData[41])-50;	//-50..200gr with 1gr/bit;
		
		BMSGet.MBMU_Status.BatteryStatus.r_MaxChargeCurrentAllowed := WORD_TO_REAL(MBMUData[42])-20000;			//-20k .. +20k A in 1A/bit steps
		BMSGet.MBMU_Status.BatteryStatus.r_MaxDischargeCurrentAllowed := WORD_TO_REAL(MBMUData[43])-20000;			//-20k .. +20k A in 1A/bit steps
		
		BMSGet.MBMU_Status.BatteryStatus.r_MaxChargePowerAllowed := WORD_TO_REAL(MBMUData[44])-20000;				//-20k .. +20k kW in 1kW/bit steps
		BMSGet.MBMU_Status.BatteryStatus.r_MaxDischargePowerAllowed := WORD_TO_REAL(MBMUData[45])-20000;			//-20k .. +20k kW in 1kW/bit steps
		
		BMSGet.MBMU_Status.BatteryStatus.r_SystemPower	:= 	WORD_TO_REAL(MBMUData[46])-20000;						//-20k .. +20k kW in 1kW/bit steps
		BMSGet.MBMU_Status.BatteryStatus.r_ChargeSOE	:=	WORD_TO_REAL(MBMUData[47])/10;
		BMSGet.MBMU_Status.BatteryStatus.r_DischargeSOE	:=	WORD_TO_REAL(MBMUData[48])/10;
		
		BMSGet.MBMU_Status.BatteryStatus.r_RemainingChargeEnergy	:=	WORD_TO_REAL(MBMUData[49]);
		BMSGet.MBMU_Status.BatteryStatus.r_RemainingDischargeEnergy	:=	WORD_TO_REAL(MBMUData[50]);
		
		BMSGet.MBMU_Status.BatteryStatus.r_MaxSystemVoltageAllowed := WORD_TO_REAL(MBMUData[51])/10; 			//0-1500V with 0.1V/bit
		BMSGet.MBMU_Status.BatteryStatus.r_MinSystemVoltageAllowed := WORD_TO_REAL(MBMUData[52])/10; 			//0-1500V with 0.1V/bit
		
		BMSGet.BattInfo := BMSGet.MBMU_Status.BatteryStatus;
		
		GetMBMUData := TRUE;
		COMretryCounter := 0;
	ELSE
		COMretryCounter := COMretryCounter +1;
		IF COMRetryCounter > 5 THEN
			b_MBComErrorActive := TRUE;
		END_IF
	END_IF
END_IF
END_METHOD

METHOD GetMBMUStaticSystemData : BOOL
VAR_INST
	MBReadBMS			: 	FB_MBReadRegs;
	DataBuffer 			: 	ARRAY[0..31] OF WORD;
	
	bCommBusy			:	BOOL;
	bComError			:	BOOL;
	errID				:	UDINT;
	cbRead				:	UDINT;
	
	TransmissionDone 	: 	f_trig;
	COMretryCounter		:	USINT := 0;
	ComTimer			:	Ton := (PT := TIME#200ms);
END_VAR

//Read ETH+MBMU SW/HW version at init.
GetMBMUStaticSystemData := FALSE;

ComTimer(in := NOT(ComTimer.Q));

MBReadBMS(
sIPAddr := Config.IP_BMS,
nTCPPort := Config.MBPort_BMS,
nUnitID := 255,//16#FF;
nMBAddr := 256,
nQuantity := 32,
cbLength := SIZEOF(DataBuffer),
pDestAddr := ADR(DataBuffer),
bExecute := ComTimer.Q,
tTimeout := T#100MS,
bBusy => bCommBusy,
bError => bComError,
nErrId => errID,
cbRead => cbRead
);

TransmissionDone(CLK := bCommBusy);

IF TransmissionDone.Q THEN
	IF NOT bComError THEN
		memcpy(destAddr := ADR(BMSGet.MBMU_Status.s_MBMU_SWVer), SrcAddr := ADR(DataBuffer[0]), n := 16);
		memcpy(destAddr  := ADR(BMSGet.MBMU_Status.s_MBMU_HWVer), SrcAddr := ADR(DataBuffer[8]), n := 16);
		memcpy(destAddr  := ADR(BMSGet.MBMU_Status.s_ETH_SWVer), SrcAddr := ADR(DataBuffer[16]), n := 16);
		memcpy(destAddr  := ADR(BMSGet.MBMU_Status.r_ETH_HWVer), SrcAddr :=ADR( DataBuffer[24]), n := 16);
		GetMBMUStaticSystemData := TRUE;
		COMretryCounter := 0;
	ELSE
		COMretryCounter := COMretryCounter +1;
		IF COMRetryCounter > 5 THEN
			b_MBComErrorActive := TRUE;
		END_IF
	END_IF
END_IF
END_METHOD

METHOD GetSBMUData : BOOL
VAR_INST
	MBReadSBMU		: 	FB_MBReadRegs;
	DataBuffer		:	ARRAY[0..87] OF WORD;
	bCommBusy		:	BOOL;
	bComError		:	BOOL;
	errID			:	UDINT;
	cbRead			:	UDINT;
	CommDone		: 	f_trig;
	
	SBMUCounter			: 	USINT	:=	0;
	COMretryCounter	:	USINT	:=	0;
	ComTimer			:	Ton := (PT := TIME#0S200MS);
END_VAR
GetSBMUData := FALSE;

ComTimer(in := NOT(ComTimer.Q));

MBReadSBMU(
	sIPAddr := Config.IP_BMS,
	nTCPPort := Config.MBPort_BMS,
	nUnitID := 255,//16#FF;
	nMBAddr := 1024*(SBMUcounter+1),
	nQuantity := 87,
	cbLength := SIZEOF(DataBuffer),
	pDestAddr := ADR(DataBuffer),
	bExecute := ComTimer.Q,
	tTimeout := TIME#100MS,
	bBusy => bCommBusy,
	bError => bComError,
	nErrId => errID,
	cbRead => cbRead
);
	
CommDone(CLK := bCommBusy);
	
IF CommDone.Q THEN
	IF NOT bComError THEN
		BMSGet.SBMU[SBMUcounter].w_SystemWarning := DataBuffer[0];
		BMSGet.SBMU[SBMUcounter].SystemAlarm[0] := DataBuffer[1];
		BMSGet.SBMU[SBMUcounter].SystemAlarm[1] := DataBuffer[2];
		BMSGet.SBMU[SBMUcounter].SystemAlarm[2] := DataBuffer[3];
		
		BMSGet.SBMU[SBMUcounter].b_PrechargeRelayClosed 	:= WORD_TO_BOOL(DataBuffer[16]);
		BMSGet.SBMU[SBMUcounter].b_MainPosRelayClosed	 	:= WORD_TO_BOOL(DataBuffer[17]);
		BMSGet.SBMU[SBMUcounter].b_MainNegRelayClosed		:= WORD_TO_BOOL(DataBuffer[18]);
		BMSGet.SBMU[SBMUcounter].b_ControlBoxFanOn 			:= WORD_TO_BOOL(DataBuffer[19]);
		BMSGet.SBMU[SBMUcounter].b_BalanceStatus 			:= WORD_TO_BOOL(DataBuffer[20]);
		
		BMSGet.SBMU[SBMUcounter].BatteryStatus.r_SystemVoltage := WORD_TO_REAL(DataBuffer[32])/10;	//0-1500V with 0.1V/bit
		BMSGet.SBMU[SBMUcounter].BatteryStatus.r_SystemCurrent := (WORD_TO_REAL(DataBuffer[34])/10)-2000; 	//-2k .. +2k A in 0.1A/bit steps
		
		BMSGet.SBMU[SBMUcounter].BatteryStatus.r_SOC := WORD_TO_REAL(DataBuffer[35])/10; 			//0-100% with 0.1%/bit;
		BMSGet.SBMU[SBMUcounter].BatteryStatus.r_SOH := WORD_TO_REAL(DataBuffer[36])/10;				//0-100% with 0.1%/bit;
		
		BMSGet.SBMU[SBMUcounter].BatteryStatus.CellVoltage[eSubValues.Maximum] := WORD_TO_REAL(DataBuffer[37])/1000;	//0-5v with 0.001v/bit;
		BMSGet.SBMU[SBMUcounter].BatteryStatus.CellVoltage[eSubValues.Average] := WORD_TO_REAL(DataBuffer[39])/1000;	//0-5v with 0.001v/bit;
		
		BMSGet.SBMU[SBMUcounter].BatteryStatus.CellTemperature[eSubValues.Maximum] := WORD_TO_REAL(DataBuffer[40])-50;	//-50..200gr with 1gr/bit;
		BMSGet.SBMU[SBMUcounter].BatteryStatus.CellTemperature[eSubValues.Minimum] := WORD_TO_REAL(DataBuffer[41])-50;	//-50..200gr with 1gr/bit;
		BMSGet.SBMU[SBMUcounter].BatteryStatus.CellTemperature[eSubValues.Average] := WORD_TO_REAL(DataBuffer[42])-50;	//-50..200gr with 1gr/bit;
		
		BMSGet.SBMU[SBMUcounter].BatteryStatus.r_MaxChargeCurrentAllowed := 		(WORD_TO_REAL(DataBuffer[43])/10)-2000;	//-2k .. +2k A in 0.1A/bit steps
		BMSGet.SBMU[SBMUcounter].BatteryStatus.r_MaxDischargeCurrentAllowed := 		(WORD_TO_REAL(DataBuffer[44])/10)-2000;	//-2k .. +2k A in 0.1A/bit steps
		
		BMSGet.SBMU[SBMUcounter].BatteryStatus.w_MaxVoltageCellLocation := DataBuffer[48];
		BMSGet.SBMU[SBMUcounter].BatteryStatus.w_MinVoltageCellLocation := DataBuffer[49];
		
		BMSGet.SBMU[SBMUcounter].BatteryStatus.w_MaxTempCellLocation := DataBuffer[50];
		BMSGet.SBMU[SBMUcounter].BatteryStatus.w_MinTempCellLocation := DataBuffer[51];
		
		BMSGet.SBMU[SBMUcounter].BatteryStatus.r_SumOfCellVoltages := WORD_TO_REAL(DataBuffer[55])/10;	//0-1500V with 0.1V/bit
		
		MEMCPY(ADR(BMSGet.SBMU[SBMUcounter].BatteryStatus.r_HistAccChargeEnergy), ADR(DataBuffer[85]), 2);  // low word
		MEMCPY(ADR(BMSGet.SBMU[SBMUcounter].BatteryStatus.r_HistAccChargeEnergy)+2, ADR(DataBuffer[84]), 2);  // high word
		BMSGet.SBMU[SBMUcounter].BatteryStatus.r_HistAccChargeEnergy := BMSGet.SBMU[SBMUcounter].BatteryStatus.r_HistAccChargeEnergy/10; //0-449GHW with 0.1kWh/bit
		
		MEMCPY(ADR(BMSGet.SBMU[SBMUcounter].BatteryStatus.r_HistAccDischargeEnergy), ADR(DataBuffer[87]), 2);  // low word
		MEMCPY(ADR(BMSGet.SBMU[SBMUcounter].BatteryStatus.r_HistAccDischargeEnergy)+2, ADR(DataBuffer[86]), 2);  // high word
		BMSGet.SBMU[SBMUcounter].BatteryStatus.r_HistAccDischargeEnergy := BMSGet.SBMU[SBMUcounter].BatteryStatus.r_HistAccDischargeEnergy/10; //0-449GHW with 0.1kWh/bit
	
		SBMUCounter := SBMUCounter +1;
		COMretryCounter := 0;
		
		IF SBMUCounter >= 4 THEN//BMSGet.MBMU_Status.by_NumberOfSubSystems THEN
			
			GetSBMUData := TRUE;
			SBMUCounter := 0;
		END_IF
		
		
		IF 		(BMSGet.SBMU[0].b_MainPosRelayClosed AND BMSGet.SBMU[0].b_MainNegRelayClosed) AND
				(BMSGet.SBMU[1].b_MainPosRelayClosed AND BMSGet.SBMU[1].b_MainNegRelayClosed) AND
				(BMSGet.SBMU[2].b_MainPosRelayClosed AND BMSGet.SBMU[2].b_MainNegRelayClosed) AND
				(BMSGet.SBMU[3].b_MainPosRelayClosed AND BMSGet.SBMU[3].b_MainNegRelayClosed) THEN
			PowerStatus := eHVDC_PowerStatus.On;
		ELSIF 	BMSGet.SBMU[SBMUcounter].b_PrechargeRelayClosed OR 
				BMSGet.SBMU[SBMUcounter].b_PrechargeRelayClosed OR 
				BMSGet.SBMU[SBMUcounter].b_PrechargeRelayClosed OR 
				BMSGet.SBMU[SBMUcounter].b_PrechargeRelayClosed THEN
			PowerStatus := eHVDC_PowerStatus.Precharging;
		ELSE
			PowerStatus := eHVDC_PowerStatus.Off;
		END_IF	
		
		BMSGet.SBMU[SBMUcounter].b_PrechargeRelayClosed 	:= WORD_TO_BOOL(DataBuffer[16]);
		BMSGet.SBMU[SBMUcounter].b_MainPosRelayClosed	 	:= WORD_TO_BOOL(DataBuffer[17]);
		BMSGet.SBMU[SBMUcounter].b_MainNegRelayClosed		:= WORD_TO_BOOL(DataBuffer[18]);
		BMSGet.SBMU[SBMUcounter].b_ControlBoxFanOn 			:= WORD_TO_BOOL(DataBuffer[19]);
		BMSGet.SBMU[SBMUcounter].b_BalanceStatus 			:= WORD_TO_BOOL(DataBuffer[20]);
	ELSE
		COMretryCounter := COMretryCounter +1;
		IF COMRetryCounter > 5 THEN
			b_MBComErrorActive := TRUE;
		END_IF
	END_IF
END_IF
END_METHOD

METHOD GetSBMUStaticSystemData : BOOL

VAR_INPUT
	SBMU_ID				:	uint;	
END_VAR

VAR_INST
	MBReadBMS			: 	FB_MBReadRegs;
	DataBuffer 			: 	ARRAY[0..31] OF WORD;
	
	bCommBusy			:	BOOL;
	bComError			:	BOOL;
	errID				:	UDINT;
	cbRead				:	UDINT;
	
	TransmissionDone 	: 	f_trig;
	ComretryCounter		:	USINT := 0;
	
	ComTimer			:	Ton := (PT := TIME#0S200MS);
END_VAR


VAR
	SBMU: INT;
END_VAR
//Read ETH+MBMU SW/HW version at init.
GetSBMUStaticSystemData := FALSE;

IF (SBMU_ID<1) OR (SBMU>4)then //BMSGET.MBMU_Status.by_NumberOfSubSystems) THEN
	GetSBMUStaticSystemData := TRUE;
	RETURN;
END_IF

ComTimer(in := NOT(ComTimer.Q));

MBReadBMS(
sIPAddr := Config.IP_BMS,
nTCPPort := Config.MBPort_BMS,
nUnitID := 255,//16#FF;
nMBAddr := 960 + (SBMU_ID*1024),
nQuantity := 32,
cbLength := SIZEOF(DataBuffer),
pDestAddr := ADR(DataBuffer),
bExecute := ComTimer.Q,
tTimeout := T#100MS,
bBusy => bCommBusy,
bError => bComError,
nErrId => errID,
cbRead => cbRead
);

TransmissionDone(CLK := bCommBusy);

IF TransmissionDone.Q THEN
	IF NOT bComError THEN
	//werkt niet. Bij de MBMU gek genoeg wel
	//	memcpy(destAddr := ADR(BMSGet.SBMU[SBMU_ID].s_SBMU_SWVer), SrcAddr := ADR(DataBuffer[0]), n := 16);
	//	memcpy(destAddr  := ADR(BMSGet.SBMU[SBMU_ID].s_SBMU_HWVer), SrcAddr := ADR(DataBuffer[8]), n := 16);
	//	memcpy(destAddr  := ADR(BMSGet.SBMU[SBMU_ID].s_CSC_SWVer), SrcAddr := ADR(DataBuffer[16]), n := 16);
	//	memcpy(destAddr  := ADR(BMSGet.SBMU[SBMU_ID].s_CSC_HWVer), SrcAddr := ADR(DataBuffer[24]), n := 16);
		GetSBMUStaticSystemData := TRUE;
		ComretryCounter := 0;
	ELSE
		COMretryCounter := COMretryCounter +1;
		IF COMRetryCounter > 5 THEN
			b_MBComErrorActive := TRUE;
		END_IF
	END_IF
END_IF
END_METHOD

METHOD GetSystemStatus : BOOL
VAR_INST
	MBReadBMS			: 	FB_MBReadRegs;
	DataBuffer 			: 	ARRAY[0..3] OF WORD;
	
	bCommBusy			:	BOOL;
	bComError			:	BOOL;
	errID				:	UDINT;
	cbRead				:	UDINT;
	
	TransmissionDone 	: 	f_trig;
	
	ComTimer			:	Ton := (PT := TIME#0S200MS);
	
	ComretryCounter	:	USINT := 0;
END_VAR

//Read general BMS status
GetSystemStatus := FALSE;

ComTimer(in := NOT(ComTimer.Q));

MBReadBMS(
sIPAddr := Config.IP_BMS,
nTCPPort := Config.MBPort_BMS,
nUnitID := 255,//16#FF;
nMBAddr := 769,
nQuantity := 4,
cbLength := SIZEOF(DataBuffer),
pDestAddr := ADR(DataBuffer),
bExecute := ComTimer.Q,
bBusy => bCommBusy,
bError => bComError,
nErrId => errID,
cbRead => cbRead,
tTimeout	:= T#100MS
);

TransmissionDone(CLK := bCommBusy);

IF TransmissionDone.Q THEN
	IF NOT bComError THEN
		CASE DataBuffer[0] OF
			0: BMSGet.MBMU_Status.BatteryStatus.ui_BMS_PowerOnStatus := ePowerOnStatus.Off;
			1: BMSGet.MBMU_Status.BatteryStatus.ui_BMS_PowerOnStatus := ePowerOnStatus.On;
			2: BMSGet.MBMU_Status.BatteryStatus.ui_BMS_PowerOnStatus := ePowerOnStatus.PowerOn_Fault;
			3: BMSGet.MBMU_Status.BatteryStatus.ui_BMS_PowerOnStatus := ePowerOnStatus.PowerOff_Fault;
		END_CASE
		
		BMSGet.BattInfo.ui_BMS_PowerOnStatus := BMSGet.MBMU_Status.BatteryStatus.ui_BMS_PowerOnStatus;
		
		CASE DataBuffer[1] OF
			0: BMSGet.MBMU_Status.BatteryStatus.ui_BMS_Status := eBMS_Status.Init;
			1: BMSGet.MBMU_Status.BatteryStatus.ui_BMS_Status := eBMS_Status.Normal;
			2: BMSGet.MBMU_Status.BatteryStatus.ui_BMS_Status := eBMS_Status.FullCharge;
			3: BMSGet.MBMU_Status.BatteryStatus.ui_BMS_Status := eBMS_Status.FullDischarge;
			4: BMSGet.MBMU_Status.BatteryStatus.ui_BMS_Status := eBMS_Status.Warning;
			5: BMSGet.MBMU_Status.BatteryStatus.ui_BMS_Status := eBMS_Status.Fault;
		END_CASE
		
		BMSGet.BattInfo.ui_BMS_Status := BMSGet.MBMU_Status.BatteryStatus.ui_BMS_Status;
		
		BMSGet.MBMU_Status.by_NumberOfSubSystems := WORD_TO_BYTE(DataBuffer[3]);
		GetSystemStatus := TRUE;
		ComretryCounter := 0;
	ELSE
		COMretryCounter := COMretryCounter +1;
		IF COMRetryCounter > 5 THEN
			b_MBComErrorActive := TRUE;
		END_IF
	END_IF
END_IF
END_METHOD

METHOD OpenInsulationSwitch : BOOL
VAR_INPUT
	OpenSwitch : BOOL;
END_VAR

VAR_INST
	WriteReg	:	FB_MBWriteSingleReg;
	Value 		:	WORD 	:= 0;
	StartWrite	:	BOOL	:= FALSE;
	
	bCommBusy	:	BOOL;
	bComError	:	BOOL;
	errID		:	UDINT;

	TransmissionDone 	: 	f_trig;
	ComRetryCounter	:	USINT;
	
	ComTimer			:	Ton := (PT := TIME#0S200MS);
END_VAR

ComTimer(in := NOT(ComTimer.Q));

OpenInsulationswitch := FALSE;

IF OpenSwitch THEN
	Value := 1;
ELSE
	Value := 0;
END_IF

WriteReg(
sIPAddr := Config.IP_BMS,
nTCPPort := Config.MBPort_BMS,
nUnitID := 255,//16#FF;
nMBAddr := 907,
nValue := Value,
tTimeout := T#0S100MS,
bExecute := ComTimer.q,
bBusy => bCommBusy,
bError => bComError,
nErrId => errID,
);

TransmissionDone(CLK := bCommBusy);

IF TransmissionDone.Q THEN
	IF NOT bComError THEN
		BMSGet.MBMU_Status.b_InsulationSwitchOpen := OpenSwitch;
		ComRetryCounter := 0;
		OpenInsulationSwitch := TRUE;
	ELSE
		COMretryCounter := COMretryCounter +1;
		IF COMRetryCounter > 5 THEN
			b_MBComErrorActive := TRUE;
		END_IF
	END_IF
END_IF
END_METHOD

METHOD Reset : BOOL
VAR_INPUT
	//BMSSET	:	st_BMS_Set;
	//ResetIn	:	BOOL;
END_VAR

VAR_INST
	ResetTrigger		:	Ton := (PT := TIME#1S0MS);
	ResetVar			:	BOOL;
END_VAR
Reset := FALSE;

IF FBState = ePOUState.Normal OR FBState = ePOUState.EMSTOP THEN
	IF ClearBMSFaults() THEN
		FBState := ePOUState.Normal;
	END_IF
END_IF
END_METHOD

METHOD SetBMSDateTime : BOOL
VAR
	SystemTimeData	:	Timestruct;
	RTCData	:	ARRAY[0..6] OF WORD;	
	
END_VAR
VAR_INST
	ComTimer			:	Ton := (PT := TIME#0S200MS);
	WriteRegs		:	FB_MBWriteRegs;
	SystemTime		:	FB_LocalSystemTime;
	TransmissionDone 	: 	f_trig;
	SystemTimeDataValid	:	BOOL;
	bCommBusy		:	BOOL;
	bComError		:	BOOL;
	errID			:	UDINT;
	COMRetryCounter	:	USINT := 0;
END_VAR
ComTimer(in := NOT(ComTimer.Q));

//write PLC system time to BMS RTC
SetBMSDateTime := FALSE;


//retrieve system time struct
SystemTime(
	sNetID := '',
	bEnable := TRUE,
	dwCycle := 1,
	dwOpt	:= 1,
	tTimeout := TIME#500MS,
	bValid => SystemtimeDataValid,
	systemTime => SystemTimeData
);

//parse system time to BMS data array
IF SystemTimeDataValid THEN
	RTCData[0] := 2024;//SystemTimeData.wYear;
	RTCData[1] := 03;//SystemTimeData.wMonth;
	RTCData[2] := 26;//SystemTimeData.wDay;
	RTCData[3] := 13;//SystemTimeData.wHour;
	RTCData[4] := 52;//SystemTimeData.wMinute;
	RTCData[5] := 00;//SystemTimeData.wSecond;
	RTCData[6] := 1;//can this value remain at 1? or reset to 0 after write?
	
	//write data to BMS
	WriteRegs(	
	sIPAddr := Config.IP_BMS,
	nTCPPort := Config.MBPort_BMS,
	nUnitID := 255,//16#FF;
	nMBAddr := 900,
	nQuantity := 7,
	pSrcAddr := ADR(RTCData),
	cbLength := SIZEOF(RTCData),
	bExecute := ComTimer.Q,
	tTimeout := TIME#100MS,
	bBusy => bCommBusy,
	bError => bComError,
	nErrId => errID,
	);
	
	TransmissionDone(CLK := bCommBusy);
	
	//return true if tranmission succeeds
	IF TransmissionDone.Q THEN
		IF NOT bComError THEN
			SetBMSDateTime := TRUE;
			ComRetryCounter := 0;
		ELSE
			COMretryCounter := COMretryCounter +1;
			IF COMRetryCounter > 5 THEN
				b_MBComErrorActive := TRUE;
			END_IF
		END_IF
	END_IF
END_IF
END_METHOD

